C03601=1034.717,46.455,-90.669,168.917,41.159,157.714
C03602=1034.724,46.704,-90.686,168.919,41.158,157.713
C03603=1034.729,46.954,-90.702,168.921,41.158,157.714
C03604=1034.735,47.203,-90.720,168.923,41.158,157.714
C03605=1034.742,47.452,-90.737,168.926,41.157,157.714
C03606=1034.748,47.701,-90.753,168.928,41.156,157.714
C03607=1034.754,47.951,-90.771,168.930,41.156,157.714
C03608=1034.760,48.200,-90.788,168.932,41.156,157.714
C03609=1034.767,48.450,-90.805,168.934,41.156,157.714
C03610=1034.773,48.699,-90.822,168.937,41.155,157.714
C03611=1034.779,48.948,-90.840,168.939,41.154,157.714
C03612=1034.785,49.198,-90.856,168.941,41.154,157.714
C03613=1034.791,49.447,-90.873,168.943,41.154,157.714
C03614=1034.797,49.696,-90.891,168.945,41.153,157.714
C03615=1034.804,49.945,-90.908,168.947,41.153,157.714
C03616=1034.810,50.195,-90.925,168.950,41.152,157.714
C03617=1034.816,50.444,-90.942,168.951,41.151,157.714
C03618=1034.823,50.694,-90.960,168.953,41.151,157.714
C03619=1034.829,50.942,-90.977,168.956,41.151,157.714
C03620=1034.835,51.192,-90.993,168.958,41.151,157.714
C03621=1034.841,51.441,-91.011,168.960,41.150,157.714
C03622=1034.848,51.691,-91.028,168.962,41.149,157.714
C03623=1034.854,51.940,-91.045,168.964,41.149,157.714
C03624=1034.860,52.190,-91.062,168.966,41.148,157.714
C03625=1034.867,52.439,-91.080,168.968,41.148,157.714
C03626=1034.873,52.688,-91.097,168.971,41.148,157.714
C03627=1034.879,52.938,-91.115,168.973,41.147,157.714
C03628=1034.885,53.187,-91.131,168.975,41.147,157.714
C03629=1034.892,53.437,-91.148,168.977,41.146,157.714
C03630=1034.897,53.686,-91.166,168.979,41.146,157.714
C03631=1034.904,53.935,-91.183,168.982,41.145,157.714
C03632=1034.911,54.184,-91.200,168.984,41.145,157.714
C03633=1034.917,54.433,-91.218,168.986,41.145,157.715
C03634=1034.923,54.682,-91.235,168.988,41.144,157.714
C03635=1034.929,54.932,-91.252,168.990,41.143,157.715
C03636=1034.936,55.182,-91.269,168.993,41.143,157.715
C03637=1034.942,55.431,-91.286,168.995,41.142,157.715
C03638=1034.949,55.680,-91.304,168.997,41.142,157.715
C03639=1034.955,55.929,-91.321,168.999,41.142,157.715
C03640=1034.961,56.179,-91.339,169.001,41.141,157.715
C03641=1034.968,56.428,-91.356,169.004,41.140,157.715
C03642=1034.974,56.677,-91.373,169.006,41.140,157.715
C03643=1034.980,56.927,-91.390,169.008,41.139,157.715
C03644=1034.986,57.176,-91.407,169.010,41.139,157.715
C03645=1034.993,57.425,-91.424,169.012,41.139,157.715
C03646=1034.999,57.675,-91.442,169.015,41.138,157.715
C03647=1035.006,57.924,-91.459,169.017,41.138,157.715
C03648=1035.012,58.174,-91.477,169.019,41.137,157.715
C03649=1035.018,58.423,-91.495,169.021,41.136,157.715
C03650=1035.025,58.672,-91.512,169.023,41.136,157.715
C03651=1035.031,58.921,-91.530,169.026,41.136,157.715
C03652=1035.038,59.171,-91.547,169.028,41.135,157.715
C03653=1035.044,59.420,-91.564,169.030,41.135,157.715
C03654=1035.050,59.669,-91.582,169.032,41.134,157.715
C03655=1035.056,59.918,-91.599,169.034,41.134,157.715
C03656=1035.064,60.205,-91.619,169.037,41.133,157.715
C03657=1035.071,60.491,-91.639,169.039,41.132,157.715
C03658=1035.079,60.777,-91.659,169.041,41.132,157.715
C03659=1035.086,61.063,-91.679,169.044,41.131,157.715
C03660=1035.092,61.313,-91.697,169.046,41.131,157.715
C03661=1035.099,61.561,-91.714,169.048,41.130,157.715
C03662=1035.105,61.811,-91.731,169.050,41.130,157.715
C03663=1035.112,62.061,-91.749,169.052,41.129,157.715
C03664=1035.118,62.310,-91.766,169.055,41.128,157.715
C03665=1035.125,62.558,-91.784,169.057,41.128,157.715
C03666=1035.131,62.808,-91.802,169.059,41.128,157.715
C03667=1035.138,63.057,-91.819,169.061,41.127,157.715
C03668=1035.144,63.306,-91.836,169.064,41.127,157.715
C03669=1035.150,63.556,-91.854,169.066,41.126,157.715
C03670=1035.157,63.805,-91.871,169.068,41.125,157.715
C03671=1035.163,64.055,-91.889,169.070,41.125,157.715
C03672=1035.169,64.304,-91.907,169.072,41.125,157.715
C03673=1035.176,64.553,-91.925,169.074,41.124,157.715
C03674=1035.182,64.802,-91.943,169.077,41.124,157.715
C03675=1035.188,65.052,-91.961,169.079,41.123,157.715
C03676=1035.194,65.301,-91.978,169.081,41.123,157.716
C03677=1035.201,65.551,-91.996,169.083,41.122,157.715
C03678=1035.208,65.800,-92.014,169.085,41.122,157.716
C03679=1035.213,66.049,-92.031,169.088,41.122,157.716
C03680=1035.219,66.298,-92.049,169.090,41.122,157.716
C03681=1035.226,66.548,-92.067,169.092,41.121,157.716
C03682=1035.232,66.796,-92.085,169.094,41.120,157.716
C03683=1035.238,67.046,-92.103,169.096,41.120,157.716
C03684=1035.245,67.295,-92.120,169.098,41.120,157.716
C03685=1035.251,67.544,-92.139,169.101,41.119,157.716
C03686=1035.257,67.793,-92.156,169.103,41.119,157.716
C03687=1035.263,68.043,-92.174,169.105,41.118,157.716
C03688=1035.270,68.292,-92.192,169.107,41.118,157.716
C03689=1035.276,68.542,-92.210,169.109,41.117,157.716
C03690=1035.282,68.791,-92.228,169.111,41.117,157.716
C03691=1035.289,69.040,-92.246,169.114,41.117,157.716
C03692=1035.295,69.289,-92.264,169.116,41.116,157.716
C03693=1035.301,69.539,-92.282,169.118,41.116,157.716
C03694=1035.308,69.788,-92.300,169.120,41.115,157.716
C03695=1035.313,70.037,-92.318,169.122,41.115,157.716
C03696=1035.320,70.287,-92.335,169.124,41.115,157.716
C03697=1035.327,70.536,-92.354,169.127,41.114,157.716
C03698=1035.333,70.786,-92.372,169.129,41.114,157.716
C03699=1035.338,71.034,-92.390,169.131,41.113,157.716
C03700=1035.345,71.284,-92.408,169.133,41.113,157.716
C03701=1035.351,71.533,-92.427,169.135,41.113,157.716
C03702=1035.357,71.783,-92.445,169.137,41.113,157.716
C03703=1035.364,72.031,-92.463,169.140,41.112,157.717
C03704=1035.370,72.280,-92.480,169.142,41.111,157.716
C03705=1035.376,72.530,-92.498,169.144,41.111,157.717
C03706=1035.382,72.779,-92.517,169.146,41.111,157.717
C03707=1035.388,73.029,-92.535,169.148,41.111,157.717
C03708=1035.395,73.278,-92.554,169.150,41.110,157.717
C03709=1035.400,73.527,-92.571,169.152,41.110,157.717
C03710=1035.408,73.776,-92.589,169.155,41.109,157.717
C03711=1035.414,74.025,-92.608,169.157,41.109,157.717
C03712=1035.420,74.275,-92.626,169.159,41.109,157.717
C03713=1035.427,74.524,-92.644,169.161,41.108,157.717
C03714=1035.433,74.774,-92.662,169.163,41.108,157.717
C03715=1035.439,75.022,-92.681,169.165,41.107,157.717
C03716=1035.445,75.272,-92.699,169.168,41.107,157.717
C03717=1035.451,75.521,-92.717,169.170,41.107,157.717
C03718=1035.457,75.771,-92.735,169.172,41.106,157.717
C03719=1035.464,76.020,-92.753,169.174,41.106,157.717
C03720=1035.471,76.305,-92.774,169.177,41.105,157.717
C03721=1035.479,76.591,-92.795,169.179,41.105,157.717
C03722=1035.485,76.877,-92.816,169.182,41.104,157.717
C03723=1035.493,77.163,-92.837,169.184,41.104,157.717
C03724=1035.499,77.413,-92.856,169.186,41.103,157.717
C03725=1035.506,77.662,-92.874,169.188,41.103,157.717
C03726=1035.511,77.911,-92.892,169.191,41.103,157.717
C03727=1035.518,78.160,-92.911,169.193,41.103,157.717
C03728=1035.524,78.409,-92.929,169.195,41.102,157.717
C03729=1035.530,78.659,-92.947,169.197,41.102,157.717
C03730=1035.536,78.908,-92.966,169.199,41.101,157.718
C03731=1035.542,79.157,-92.985,169.201,41.101,157.718
C03732=1035.548,79.407,-93.003,169.203,41.101,157.718
C03733=1035.555,79.656,-93.022,169.206,41.100,157.718
C03734=1035.561,79.905,-93.040,169.208,41.100,157.718
C03735=1035.567,80.154,-93.059,169.210,41.100,157.718
C03736=1035.573,80.403,-93.077,169.212,41.100,157.718
C03737=1035.579,80.653,-93.096,169.214,41.099,157.718
C03738=1035.585,80.902,-93.114,169.216,41.099,157.718
C03739=1035.592,81.151,-93.133,169.218,41.098,157.718
C03740=1035.598,81.400,-93.152,169.221,41.098,157.718
C03741=1035.604,81.650,-93.170,169.223,41.098,157.718
C03742=1035.611,81.899,-93.188,169.225,41.097,157.718
C03743=1035.616,82.149,-93.208,169.227,41.097,157.718
C03744=1035.623,82.398,-93.226,169.229,41.097,157.718
C03745=1035.629,82.646,-93.244,169.231,41.096,157.718
C03746=1035.635,82.895,-93.263,169.233,41.096,157.718
C03747=1035.641,83.145,-93.281,169.236,41.096,157.718
C03748=1035.648,83.394,-93.300,169.238,41.095,157.718
C03749=1035.653,83.643,-93.319,169.240,41.095,157.719
C03750=1035.660,83.893,-93.338,169.242,41.095,157.719
C03751=1035.666,84.142,-93.356,169.244,41.095,157.719
C03752=1035.673,84.391,-93.375,169.246,41.094,157.719
C03753=1035.679,84.640,-93.394,169.249,41.093,157.719
C03754=1035.685,84.889,-93.412,169.251,41.093,157.719
C03755=1035.691,85.139,-93.431,169.253,41.093,157.719
C03756=1035.697,85.388,-93.449,169.255,41.093,157.719
C03757=1035.704,85.637,-93.468,169.257,41.092,157.719
C03758=1035.710,85.887,-93.487,169.259,41.091,157.719
C03759=1035.717,86.136,-93.505,169.262,41.091,157.719
C03760=1035.722,86.385,-93.525,169.264,41.091,157.719
C03761=1035.729,86.634,-93.543,169.266,41.091,157.719
C03762=1035.735,86.883,-93.562,169.268,41.090,157.719
C03763=1035.742,87.132,-93.580,169.270,41.090,157.719
C03764=1035.748,87.382,-93.599,169.272,41.089,157.719
C03765=1035.754,87.631,-93.618,169.275,41.089,157.719
C03766=1035.760,87.880,-93.637,169.277,41.089,157.719
C03767=1035.766,88.129,-93.656,169.279,41.088,157.719
C03768=1035.773,88.378,-93.674,169.281,41.088,157.719
C03769=1035.779,88.627,-93.693,169.283,41.087,157.719
C03770=1035.786,88.877,-93.712,169.286,41.087,157.719
C03771=1035.791,89.126,-93.731,169.288,41.087,157.719
C03772=1035.798,89.375,-93.750,169.290,41.086,157.719
C03773=1035.805,89.625,-93.769,169.292,41.086,157.720
C03774=1035.811,89.874,-93.787,169.294,41.085,157.719
C03775=1035.817,90.124,-93.806,169.296,41.085,157.720
C03776=1035.823,90.373,-93.825,169.299,41.085,157.720
C03777=1035.829,90.622,-93.844,169.301,41.084,157.720
C03778=1035.836,90.871,-93.864,169.303,41.084,157.720
C03779=1035.842,91.120,-93.883,169.305,41.084,157.720
C03780=1035.848,91.369,-93.902,169.307,41.084,157.720
C03781=1035.854,91.619,-93.921,169.309,41.084,157.720
C03782=1035.860,91.868,-93.939,169.311,41.083,157.720
C03783=1035.867,92.117,-93.958,169.314,41.083,157.720
C03784=1035.874,92.403,-93.980,169.316,41.083,157.720
C03785=1035.880,92.688,-94.002,169.319,41.082,157.720
C03786=1035.887,92.974,-94.025,169.321,41.082,157.720
C03787=1035.894,93.260,-94.046,169.324,41.082,157.720
C03788=1035.901,93.509,-94.066,169.326,41.081,157.720
C03789=1035.907,93.758,-94.085,169.328,41.081,157.721
C03790=1035.913,94.008,-94.104,169.330,41.080,157.720
C03791=1035.919,94.257,-94.123,169.332,41.080,157.720
C03792=1035.926,94.505,-94.142,169.334,41.080,157.721
C03793=1035.931,94.755,-94.161,169.336,41.080,157.721
C03794=1035.938,95.004,-94.180,169.339,41.079,157.721
C03795=1035.944,95.254,-94.200,169.341,41.079,157.721
C03796=1035.951,95.503,-94.219,169.343,41.079,157.721
C03797=1035.956,95.752,-94.238,169.345,41.079,157.721
C03798=1035.963,96.001,-94.257,169.347,41.078,157.721
C03799=1035.969,96.251,-94.276,169.349,41.078,157.721
C03800=1035.975,96.499,-94.296,169.352,41.078,157.721
C03801=1035.981,96.749,-94.315,169.354,41.077,157.721
C03802=1035.987,96.998,-94.333,169.356,41.077,157.721
C03803=1035.994,97.247,-94.354,169.358,41.076,157.721
C03804=1036.000,97.496,-94.372,169.360,41.076,157.721
C03805=1036.006,97.746,-94.392,169.363,41.076,157.721
C03806=1036.013,97.994,-94.411,169.365,41.076,157.721
C03807=1036.018,98.244,-94.430,169.367,41.075,157.721
C03808=1036.025,98.493,-94.449,169.369,41.075,157.721
C03809=1036.032,98.742,-94.469,169.371,41.075,157.722
C03810=1036.038,98.991,-94.488,169.373,41.075,157.722
C03811=1036.044,99.240,-94.508,169.376,41.074,157.722
C03812=1036.050,99.489,-94.526,169.378,41.073,157.722
C03813=1036.056,99.739,-94.546,169.380,41.073,157.722
C03814=1036.063,99.988,-94.565,169.382,41.073,157.722
C03815=1036.069,100.237,-94.585,169.384,41.073,157.722
C03816=1036.075,100.486,-94.605,169.387,41.072,157.722
C03817=1036.081,100.735,-94.623,169.389,41.072,157.722
C03818=1036.087,100.984,-94.643,169.391,41.072,157.722
C03819=1036.093,101.234,-94.662,169.393,41.071,157.722
C03820=1036.100,101.483,-94.683,169.395,41.071,157.722
C03821=1036.106,101.732,-94.701,169.397,41.071,157.722
C03822=1036.112,101.981,-94.721,169.400,41.071,157.722
C03823=1036.118,102.231,-94.741,169.402,41.070,157.722
C03824=1036.124,102.479,-94.761,169.404,41.070,157.722
C03825=1036.130,102.729,-94.780,169.406,41.070,157.722
C03826=1036.137,102.978,-94.800,169.408,41.070,157.722
C03827=1036.143,103.227,-94.820,169.411,41.069,157.723
C03828=1036.149,103.476,-94.839,169.414,41.069,157.723
C03829=1036.155,103.725,-94.859,169.416,41.069,157.723
C03830=1036.161,103.974,-94.877,169.418,41.069,157.723
C03831=1036.168,104.224,-94.898,169.420,41.068,157.723
C03832=1036.174,104.472,-94.918,169.422,41.068,157.723
C03833=1036.179,104.722,-94.937,169.424,41.068,157.723
C03834=1036.185,104.971,-94.957,169.427,41.068,157.723
C03835=1036.192,105.221,-94.976,169.429,41.067,157.723
C03836=1036.198,105.469,-94.996,169.431,41.067,157.723
C03837=1036.204,105.718,-95.016,169.433,41.067,157.723
C03838=1036.210,105.968,-95.035,169.435,41.067,157.723
C03839=1036.217,106.217,-95.055,169.438,41.066,157.723
C03840=1036.223,106.466,-95.075,169.440,41.066,157.723
C03841=1036.229,106.715,-95.094,169.442,41.066,157.723
C03842=1036.235,106.964,-95.114,169.444,41.066,157.724
C03843=1036.242,107.213,-95.134,169.446,41.065,157.724
C03844=1036.247,107.463,-95.154,169.448,41.065,157.724
C03845=1036.254,107.711,-95.173,169.451,41.065,157.724
C03846=1036.261,107.961,-95.193,169.453,41.064,157.724
C03847=1036.267,108.210,-95.213,169.455,41.064,157.724
C03848=1036.274,108.495,-95.236,169.458,41.064,157.724
C03849=1036.281,108.781,-95.258,169.460,41.064,157.724
C03850=1036.288,109.067,-95.281,169.463,41.063,157.724
C03851=1036.295,109.353,-95.304,169.465,41.063,157.724
C03852=1036.301,109.602,-95.324,169.467,41.063,157.724
C03853=1036.308,109.852,-95.343,169.470,41.062,157.724
C03854=1036.314,110.101,-95.363,169.472,41.062,157.724
C03855=1036.320,110.349,-95.383,169.474,41.062,157.724
C03856=1036.326,110.599,-95.403,169.476,41.062,157.724
C03857=1036.332,110.848,-95.423,169.478,41.061,157.725
C03858=1036.338,111.097,-95.442,169.481,41.061,157.725
C03859=1036.345,111.347,-95.462,169.483,41.061,157.725
C03860=1036.351,111.595,-95.482,169.485,41.061,157.725
C03861=1036.357,111.844,-95.502,169.487,41.060,157.725
C03862=1036.363,112.094,-95.523,169.489,41.060,157.725
C03863=1036.369,112.343,-95.543,169.492,41.060,157.725
C03864=1036.375,112.591,-95.563,169.495,41.060,157.725
C03865=1036.382,112.841,-95.583,169.497,41.059,157.725
C03866=1036.388,113.090,-95.602,169.499,41.059,157.725
C03867=1036.394,113.340,-95.623,169.501,41.059,157.725
C03868=1036.400,113.589,-95.642,169.504,41.058,157.725
C03869=1036.406,113.837,-95.662,169.506,41.058,157.725
C03870=1036.412,114.087,-95.683,169.508,41.058,157.725
C03871=1036.418,114.336,-95.703,169.510,41.058,157.726
C03872=1036.424,114.585,-95.723,169.512,41.058,157.726
C03873=1036.430,114.834,-95.743,169.515,41.058,157.726
C03874=1036.436,115.084,-95.764,169.517,41.058,157.726
C03875=1036.442,115.332,-95.784,169.519,41.057,157.726
C03876=1036.449,115.581,-95.805,169.521,41.057,157.726
C03877=1036.455,115.830,-95.825,169.523,41.057,157.726
C03878=1036.460,116.079,-95.846,169.525,41.057,157.726
C03879=1036.467,116.329,-95.866,169.528,41.057,157.726
C03880=1036.473,116.578,-95.886,169.530,41.057,157.726
C03881=1036.479,116.826,-95.906,169.532,41.056,157.726
C03882=1036.484,117.076,-95.927,169.534,41.056,157.726
C03883=1036.490,117.325,-95.947,169.536,41.057,157.727
C03884=1036.496,117.574,-95.967,169.540,41.056,157.727
C03885=1036.503,117.823,-95.987,169.542,41.056,157.727
C03886=1036.508,118.072,-96.008,169.544,41.056,157.727
C03887=1036.515,118.321,-96.029,169.546,41.055,157.727
C03888=1036.521,118.570,-96.049,169.548,41.055,157.727
C03889=1036.527,118.819,-96.069,169.551,41.055,157.727
C03890=1036.533,119.069,-96.090,169.553,41.055,157.727
C03891=1036.539,119.318,-96.109,169.555,41.055,157.727
C03892=1036.546,119.567,-96.130,169.557,41.055,157.727
C03893=1036.552,119.815,-96.150,169.559,41.055,157.727
C03894=1036.558,120.065,-96.171,169.562,41.054,157.727
C03895=1036.564,120.314,-96.191,169.564,41.054,157.728
C03896=1036.570,120.563,-96.212,169.566,41.054,157.728
C03897=1036.576,120.813,-96.232,169.568,41.053,157.728
C03898=1036.582,121.061,-96.253,169.571,41.054,157.728
C03899=1036.589,121.310,-96.273,169.573,41.054,157.728
C03900=1036.595,121.559,-96.293,169.575,41.053,157.728
C03901=1036.600,121.809,-96.314,169.577,41.053,157.728
C03902=1036.606,122.058,-96.334,169.579,41.053,157.728
C03903=1036.613,122.307,-96.355,169.582,41.052,157.728
C03904=1036.619,122.556,-96.376,169.584,41.052,157.728
C03905=1036.625,122.805,-96.396,169.586,41.052,157.728
C03906=1036.631,123.053,-96.417,169.589,41.052,157.729
C03907=1036.638,123.303,-96.437,169.592,41.052,157.729
C03908=1036.643,123.552,-96.458,169.594,41.052,157.729
C03909=1036.650,123.802,-96.478,169.596,41.052,157.729
C03910=1036.656,124.050,-96.499,169.598,41.051,157.729
C03911=1036.662,124.300,-96.519,169.601,41.051,157.729
C03912=1036.669,124.585,-96.543,169.603,41.051,157.729
C03913=1036.676,124.870,-96.567,169.606,41.050,157.729
C03914=1036.683,125.156,-96.590,169.608,41.051,157.729
C03915=1036.690,125.443,-96.614,169.611,41.050,157.729
C03916=1036.697,125.691,-96.634,169.613,41.050,157.729
C03917=1036.703,125.940,-96.655,169.615,41.050,157.729
C03918=1036.709,126.189,-96.675,169.618,41.050,157.729
C03919=1036.715,126.438,-96.696,169.620,41.049,157.730
C03920=1036.722,126.688,-96.717,169.622,41.049,157.730
C03921=1036.728,126.936,-96.737,169.625,41.049,157.730
C03922=1036.734,127.186,-96.758,169.627,41.048,157.730
C03923=1036.740,127.435,-96.778,169.629,41.048,157.730
C03924=1036.747,127.684,-96.799,169.631,41.049,157.730
C03925=1036.752,127.933,-96.820,169.634,41.048,157.730
C03926=1036.759,128.182,-96.841,169.636,41.048,157.730
C03927=1036.766,128.431,-96.861,169.638,41.048,157.730
C03928=1036.771,128.680,-96.882,169.642,41.047,157.730
C03929=1036.778,128.929,-96.903,169.644,41.047,157.730
C03930=1036.785,129.179,-96.923,169.646,41.047,157.730
C03931=1036.790,129.427,-96.944,169.648,41.047,157.730
C03932=1036.797,129.677,-96.965,169.651,41.046,157.731
C03933=1036.803,129.925,-96.985,169.653,41.046,157.731
C03934=1036.809,130.175,-97.006,169.655,41.046,157.731
C03935=1036.816,130.424,-97.027,169.658,41.046,157.731
C03936=1036.822,130.672,-97.047,169.660,41.046,157.731
C03937=1036.828,130.922,-97.069,169.662,41.046,157.731
C03938=1036.835,131.170,-97.090,169.664,41.045,157.731
C03939=1036.840,131.420,-97.111,169.667,41.045,157.731
C03940=1036.846,131.669,-97.132,169.669,41.045,157.731
C03941=1036.852,131.918,-97.152,169.671,41.045,157.731
C03942=1036.858,132.167,-97.174,169.673,41.045,157.731
C03943=1036.865,132.416,-97.195,169.676,41.045,157.732
C03944=1036.871,132.665,-97.215,169.678,41.044,157.732
C03945=1036.877,132.914,-97.237,169.680,41.045,157.732
C03946=1036.884,133.163,-97.258,169.683,41.044,157.732
C03947=1036.889,133.412,-97.279,169.685,41.044,157.732
C03948=1036.895,133.661,-97.300,169.688,41.044,157.732
C03949=1036.901,133.909,-97.321,169.690,41.044,157.732
C03950=1036.907,134.159,-97.342,169.693,41.044,157.732
C03951=1036.913,134.408,-97.363,169.695,41.044,157.732
C03952=1036.920,134.657,-97.384,169.697,41.043,157.732
C03953=1036.926,134.906,-97.406,169.700,41.044,157.733
C03954=1036.932,135.156,-97.427,169.702,41.044,157.733
C03955=1036.938,135.404,-97.447,169.704,41.043,157.733
C03956=1036.944,135.653,-97.469,169.706,41.043,157.733
C03957=1036.951,135.902,-97.490,169.709,41.043,157.733
C03958=1036.957,136.152,-97.511,169.711,41.043,157.733
C03959=1036.962,136.400,-97.532,169.713,41.043,157.733
C03960=1036.969,136.649,-97.553,169.716,41.042,157.733
C03961=1036.976,136.898,-97.575,169.719,41.043,157.733
C03962=1036.981,137.147,-97.596,169.721,41.043,157.733
C03963=1036.987,137.397,-97.617,169.724,41.042,157.734
C03964=1036.994,137.646,-97.638,169.726,41.042,157.734
C03965=1036.999,137.894,-97.659,169.728,41.042,157.734
C03966=1037.006,138.143,-97.681,169.730,41.042,157.734
C03967=1037.012,138.393,-97.703,169.733,41.042,157.734
C03968=1037.019,138.641,-97.724,169.735,41.042,157.734
C03969=1037.024,138.891,-97.744,169.737,41.042,157.734
C03970=1037.030,139.140,-97.766,169.740,41.042,157.734
C03971=1037.036,139.389,-97.788,169.742,41.041,157.734
C03972=1037.042,139.638,-97.809,169.744,41.042,157.735
C03973=1037.049,139.886,-97.830,169.747,41.041,157.735
C03974=1037.055,140.136,-97.851,169.749,41.041,157.735
C03975=1037.061,140.385,-97.873,169.752,41.042,157.735
C03976=1037.068,140.670,-97.898,169.755,41.041,157.735
C03977=1037.075,140.955,-97.922,169.758,41.042,157.735
C03978=1037.082,141.241,-97.947,169.760,41.041,157.735
C03979=1037.088,141.526,-97.972,169.763,41.041,157.735
C03980=1037.095,141.775,-97.994,169.765,41.041,157.736
C03981=1037.101,142.025,-98.015,169.767,41.041,157.736
C03982=1037.108,142.273,-98.036,169.770,41.041,157.736
C03983=1037.113,142.522,-98.058,169.772,41.041,157.736
C03984=1037.119,142.771,-98.079,169.774,41.041,157.736
C03985=1037.125,143.020,-98.101,169.777,41.041,157.736
C03986=1037.132,143.270,-98.122,169.780,41.041,157.736
C03987=1037.137,143.518,-98.144,169.782,41.041,157.736
C03988=1037.143,143.767,-98.165,169.785,41.041,157.736
C03989=1037.150,144.016,-98.187,169.787,41.041,157.737
C03990=1037.156,144.266,-98.209,169.789,41.040,157.737
C03991=1037.162,144.515,-98.230,169.792,41.041,157.737
C03992=1037.168,144.764,-98.252,169.794,41.041,157.737
C03993=1037.174,145.012,-98.274,169.797,41.040,157.737
C03994=1037.181,145.261,-98.295,169.799,41.041,157.737
C03995=1037.187,145.510,-98.317,169.801,41.040,157.737
C03996=1037.193,145.759,-98.338,169.804,41.040,157.737
C03997=1037.199,146.008,-98.360,169.806,41.040,157.737
C03998=1037.205,146.258,-98.382,169.808,41.040,157.738
C03999=1037.211,146.506,-98.403,169.812,41.040,157.738
C04000=1037.217,146.755,-98.425,169.814,41.040,157.738
C04001=1037.224,147.004,-98.447,169.816,41.040,157.738
C04002=1037.230,147.253,-98.468,169.819,41.040,157.738
C04003=1037.236,147.502,-98.490,169.821,41.040,157.738
C04004=1037.242,147.751,-98.512,169.823,41.040,157.738
C04005=1037.249,148.000,-98.534,169.826,41.040,157.738
C04006=1037.253,148.249,-98.556,169.828,41.040,157.738
C04007=1037.260,148.498,-98.578,169.831,41.040,157.739
C04008=1037.266,148.747,-98.600,169.833,41.040,157.739
C04009=1037.272,148.996,-98.622,169.836,41.040,157.739
C04010=1037.278,149.245,-98.643,169.839,41.040,157.739
C04011=1037.285,149.494,-98.665,169.841,41.040,157.739
C04012=1037.291,149.743,-98.687,169.843,41.040,157.739
C04013=1037.296,149.993,-98.709,169.846,41.040,157.739
C04014=1037.302,150.240,-98.731,169.848,41.040,157.740
C04015=1037.308,150.490,-98.753,169.850,41.040,157.740
C04016=1037.315,150.739,-98.775,169.853,41.040,157.740
C04017=1037.321,150.987,-98.797,169.855,41.040,157.740
C04018=1037.327,151.237,-98.819,169.859,41.040,157.740
C04019=1037.333,151.485,-98.842,169.861,41.040,157.740
C04020=1037.339,151.735,-98.863,169.863,41.040,157.740
C04021=1037.345,151.984,-98.885,169.866,41.040,157.740
C04022=1037.352,152.232,-98.907,169.868,41.040,157.741
C04023=1037.358,152.482,-98.929,169.870,41.040,157.741
C04024=1037.364,152.731,-98.952,169.873,41.040,157.741
C04025=1037.370,152.980,-98.973,169.875,41.040,157.741
C04026=1037.376,153.228,-98.995,169.878,41.040,157.741
C04027=1037.382,153.477,-99.017,169.880,41.040,157.741
C04028=1037.388,153.726,-99.039,169.883,41.041,157.741
C04029=1037.394,153.975,-99.062,169.886,41.040,157.742
C04030=1037.400,154.224,-99.083,169.888,41.040,157.742
C04031=1037.406,154.473,-99.106,169.891,41.040,157.742
C04032=1037.414,154.794,-99.134,169.894,41.040,157.742
C04033=1037.422,155.115,-99.164,169.897,41.040,157.742
C04034=1037.430,155.437,-99.192,169.900,41.040,157.742
C04035=1037.438,155.758,-99.220,169.903,41.041,157.743
C04036=1037.443,155.989,-99.241,169.905,41.040,157.743
C04037=1037.449,156.219,-99.262,169.909,41.041,157.743
C04038=1037.454,156.450,-99.282,169.911,41.040,157.743
C04039=1037.460,156.682,-99.303,169.913,41.041,157.743
C04040=1037.466,156.912,-99.324,169.915,41.041,157.743
C04041=1037.471,157.143,-99.344,169.917,41.041,157.743
C04042=1037.478,157.374,-99.365,169.920,41.041,157.743
C04043=1037.483,157.605,-99.386,169.922,41.041,157.744
C04044=1037.489,157.854,-99.408,169.924,41.041,157.744
C04045=1037.495,158.103,-99.431,169.928,41.041,157.744
C04046=1037.501,158.351,-99.453,169.930,41.041,157.744
C04047=1037.507,158.601,-99.475,169.933,41.041,157.744
C04048=1037.513,158.850,-99.498,169.935,41.042,157.744
C04049=1037.520,159.098,-99.520,169.938,41.041,157.744
C04050=1037.525,159.348,-99.542,169.940,41.042,157.745
C04051=1037.532,159.596,-99.564,169.942,41.041,157.745
C04052=1037.538,159.845,-99.587,169.945,41.042,157.745
C04053=1037.545,160.094,-99.610,169.947,41.041,157.745
C04054=1037.550,160.344,-99.632,169.951,41.042,157.745
C04055=1037.556,160.593,-99.655,169.953,41.042,157.745
C04056=1037.562,160.841,-99.678,169.956,41.042,157.746
C04057=1037.568,161.090,-99.701,169.958,41.043,157.746
C04058=1037.574,161.339,-99.724,169.960,41.042,157.746
C04059=1037.580,161.588,-99.746,169.963,41.043,157.746
C04060=1037.586,161.837,-99.769,169.966,41.043,157.746
C04061=1037.592,162.086,-99.792,169.969,41.043,157.747
C04062=1037.597,162.334,-99.815,169.971,41.043,157.747
C04063=1037.603,162.584,-99.837,169.973,41.044,157.747
C04064=1037.609,162.833,-99.859,169.976,41.044,157.747
C04065=1037.615,163.081,-99.882,169.978,41.044,157.747
C04066=1037.621,163.330,-99.905,169.982,41.044,157.747
C04067=1037.626,163.579,-99.928,169.984,41.044,157.747
C04068=1037.633,163.828,-99.951,169.986,41.045,157.748
C04069=1037.639,164.077,-99.973,169.989,41.045,157.748
C04070=1037.644,164.326,-99.996,169.991,41.045,157.748
C04071=1037.650,164.575,-100.019,169.994,41.046,157.748
C04072=1037.656,164.823,-100.042,169.996,41.045,157.748
C04073=1037.662,165.072,-100.065,170.000,41.046,157.749
C04074=1037.668,165.321,-100.088,170.002,41.046,157.749
C04075=1037.674,165.571,-100.111,170.005,41.046,157.749
C04076=1037.680,165.819,-100.134,170.007,41.046,157.749
C04077=1037.686,166.068,-100.158,170.009,41.046,157.749
C04078=1037.693,166.316,-100.180,170.012,41.047,157.749
C04079=1037.698,166.565,-100.203,170.015,41.047,157.750
C04080=1037.704,166.814,-100.226,170.018,41.047,157.750
C04081=1037.710,167.063,-100.249,170.020,41.047,157.750
C04082=1037.715,167.312,-100.272,170.023,41.047,157.750
C04083=1037.723,167.561,-100.294,170.025,41.048,157.750
C04084=1037.728,167.810,-100.317,170.028,41.048,157.751
C04085=1037.734,168.059,-100.340,170.031,41.048,157.751
C04086=1037.740,168.308,-100.363,170.034,41.048,157.751
C04087=1037.746,168.556,-100.387,170.036,41.048,157.751
C04088=1037.752,168.805,-100.409,170.039,41.049,157.751
C04089=1037.759,169.054,-100.433,170.041,41.049,157.751
C04090=1037.764,169.303,-100.455,170.044,41.049,157.752
C04091=1037.770,169.552,-100.478,170.046,41.049,157.752
C04092=1037.776,169.800,-100.502,170.050,41.049,157.752
C04093=1037.782,170.049,-100.525,170.052,41.050,157.752
C04094=1037.789,170.299,-100.548,170.055,41.050,157.752
C04095=1037.795,170.547,-100.571,170.057,41.051,157.753
C04096=1037.800,170.796,-100.594,170.060,41.051,157.753
C04097=1037.806,171.045,-100.617,170.062,41.051,157.753
C04098=1037.812,171.294,-100.640,170.066,41.051,157.753
C04099=1037.818,171.543,-100.664,170.068,41.051,157.753
C04100=1037.825,171.792,-100.686,170.071,41.051,157.753
C04101=1037.831,172.040,-100.710,170.073,41.052,157.754
C04102=1037.837,172.290,-100.733,170.076,41.052,157.754
C04103=1037.843,172.538,-100.756,170.078,41.052,157.754
C04104=1037.850,172.822,-100.782,170.082,41.052,157.754
C04105=1037.857,173.108,-100.809,170.085,41.052,157.754
C04106=1037.864,173.392,-100.835,170.088,41.053,157.755
C04107=1037.871,173.677,-100.862,170.091,41.053,157.755
C04108=1037.877,173.925,-100.886,170.094,41.053,157.755
C04109=1037.883,174.175,-100.909,170.097,41.054,157.755
C04110=1037.890,174.424,-100.931,170.100,41.054,157.755
C04111=1037.896,174.672,-100.955,170.102,41.054,157.755
C04112=1037.901,174.921,-100.978,170.105,41.054,157.756
C04113=1037.908,175.170,-101.002,170.107,41.054,157.756
C04114=1037.914,175.419,-101.025,170.110,41.055,157.756
C04115=1037.920,175.667,-101.048,170.114,41.055,157.756
C04116=1037.926,175.916,-101.072,170.116,41.055,157.757
C04117=1037.933,176.165,-101.094,170.119,41.055,157.757
C04118=1037.939,176.414,-101.118,170.121,41.055,157.757
C04119=1037.945,176.663,-101.141,170.124,41.056,157.757
C04120=1037.951,176.911,-101.165,170.127,41.056,157.757
C04121=1037.957,177.161,-101.188,170.130,41.056,157.757
C04122=1037.963,177.409,-101.212,170.133,41.057,157.758
C04123=1037.969,177.658,-101.235,170.135,41.057,157.758
C04124=1037.977,177.907,-101.258,170.138,41.057,157.758
C04125=1037.982,178.156,-101.281,170.141,41.057,157.758
C04126=1037.989,178.405,-101.305,170.143,41.057,157.758
C04127=1037.995,178.653,-101.328,170.147,41.057,157.759
C04128=1038.001,178.902,-101.352,170.149,41.058,157.759
C04129=1038.007,179.151,-101.375,170.152,41.058,157.759
C04130=1038.013,179.400,-101.399,170.155,41.058,157.759
C04131=1038.019,179.649,-101.422,170.157,41.059,157.759
C04132=1038.025,179.897,-101.446,170.160,41.058,157.759
C04133=1038.033,180.146,-101.469,170.164,41.059,157.760
C04134=1038.039,180.395,-101.492,170.166,41.059,157.760
C04135=1038.045,180.644,-101.516,170.169,41.059,157.760
C04136=1038.051,180.893,-101.539,170.171,41.060,157.760
C04137=1038.058,181.142,-101.563,170.174,41.060,157.761
C04138=1038.064,181.390,-101.587,170.177,41.060,157.761
C04139=1038.070,181.640,-101.610,170.180,41.061,157.761
C04140=1038.076,181.888,-101.634,170.183,41.060,157.761
C04141=1038.083,182.137,-101.658,170.186,41.061,157.761
C04142=1038.088,182.386,-101.681,170.188,41.061,157.761
C04143=1038.096,182.635,-101.704,170.191,41.061,157.762
C04144=1038.102,182.883,-101.728,170.194,41.061,157.762
C04145=1038.108,183.132,-101.751,170.197,41.062,157.762
C04146=1038.114,183.381,-101.775,170.200,41.062,157.762
C04147=1038.120,183.630,-101.799,170.203,41.062,157.763
C04148=1038.126,183.878,-101.823,170.205,41.063,157.763
C04149=1038.133,184.127,-101.847,170.208,41.063,157.763
C04150=1038.138,184.376,-101.871,170.212,41.064,157.763
C04151=1038.144,184.624,-101.895,170.214,41.064,157.763
C04152=1038.150,184.873,-101.920,170.217,41.065,157.764
C04153=1038.156,185.122,-101.943,170.219,41.065,157.764
C04154=1038.162,185.372,-101.967,170.223,41.066,157.764
C04155=1038.168,185.620,-101.991,170.226,41.066,157.764
C04156=1038.173,185.869,-102.015,170.228,41.067,157.765
C04157=1038.180,186.117,-102.039,170.231,41.067,157.765
C04158=1038.185,186.367,-102.064,170.234,41.067,157.765
C04159=1038.191,186.615,-102.087,170.237,41.068,157.765
C04160=1038.197,186.864,-102.112,170.240,41.068,157.766
C04161=1038.203,187.113,-102.136,170.242,41.069,157.766
C04162=1038.209,187.362,-102.160,170.245,41.069,157.766
C04163=1038.215,187.610,-102.184,170.249,41.070,157.766
C04164=1038.222,187.859,-102.209,170.251,41.070,157.767
C04165=1038.228,188.107,-102.233,170.254,41.071,157.767
C04166=1038.233,188.356,-102.258,170.257,41.071,157.767
C04167=1038.240,188.605,-102.281,170.260,41.072,157.767
C04168=1038.247,188.889,-102.309,170.263,41.072,157.768
C04169=1038.253,189.173,-102.336,170.266,41.073,157.768
C04170=1038.260,189.458,-102.364,170.270,41.073,157.768
C04171=1038.267,189.742,-102.392,170.273,41.074,157.768
C04172=1038.273,189.991,-102.416,170.276,41.074,157.769
C04173=1038.279,190.240,-102.441,170.279,41.075,157.769
C04174=1038.285,190.488,-102.464,170.283,41.075,157.769
C04175=1038.291,190.737,-102.490,170.285,41.076,157.770
C04176=1038.298,190.986,-102.514,170.288,41.076,157.770
C04177=1038.303,191.234,-102.538,170.291,41.077,157.770
C04178=1038.310,191.483,-102.562,170.293,41.077,157.770
C04179=1038.315,191.732,-102.586,170.297,41.078,157.771
C04180=1038.322,191.980,-102.611,170.300,41.078,157.771
C04181=1038.328,192.230,-102.636,170.302,41.078,157.771
C04182=1038.334,192.478,-102.659,170.306,41.079,157.771
C04183=1038.340,192.727,-102.684,170.309,41.080,157.772
C04184=1038.347,192.976,-102.709,170.312,41.080,157.772
C04185=1038.352,193.224,-102.733,170.314,41.081,157.772
C04186=1038.359,193.473,-102.757,170.318,41.081,157.772
C04187=1038.365,193.722,-102.782,170.321,41.081,157.773
C04188=1038.371,193.970,-102.806,170.323,41.082,157.773
C04189=1038.377,194.219,-102.830,170.326,41.083,157.773
C04190=1038.384,194.468,-102.855,170.329,41.083,157.773
C04191=1038.389,194.716,-102.879,170.333,41.083,157.774
C04192=1038.396,194.965,-102.903,170.335,41.084,157.774
C04193=1038.402,195.214,-102.929,170.338,41.085,157.774
C04194=1038.409,195.463,-102.953,170.341,41.085,157.774
C04195=1038.414,195.712,-102.977,170.345,41.086,157.775
C04196=1038.420,195.960,-103.002,170.347,41.086,157.775
C04197=1038.427,196.209,-103.026,170.350,41.087,157.775
C04198=1038.432,196.457,-103.051,170.354,41.087,157.775
C04199=1038.439,196.706,-103.075,170.357,41.087,157.776
C04200=1038.445,196.955,-103.100,170.360,41.088,157.776
C04201=1038.452,197.204,-103.125,170.362,41.089,157.776
C04202=1038.458,197.453,-103.149,170.365,41.089,157.776
C04203=1038.464,197.701,-103.174,170.369,41.090,157.777
C04204=1038.470,197.950,-103.198,170.372,41.090,157.777
C04205=1038.476,198.199,-103.224,170.375,41.090,157.777
C04206=1038.483,198.448,-103.248,170.378,41.091,157.778
C04207=1038.488,198.696,-103.273,170.381,41.092,157.778
C04208=1038.495,198.945,-103.297,170.384,41.093,157.778
C04209=1038.501,199.193,-103.322,170.387,41.093,157.778
C04210=1038.508,199.442,-103.346,170.391,41.093,157.779
C04211=1038.514,199.691,-103.372,170.393,41.094,157.779
C04212=1038.521,199.940,-103.396,170.396,41.094,157.779
C04213=1038.526,200.188,-103.421,170.399,41.095,157.779
C04214=1038.533,200.437,-103.446,170.403,41.096,157.780
C04215=1038.539,200.686,-103.470,170.406,41.096,157.780
C04216=1038.545,200.934,-103.495,170.409,41.097,157.780
C04217=1038.552,201.183,-103.521,170.412,41.098,157.781
C04218=1038.557,201.432,-103.545,170.415,41.098,157.781
C04219=1038.564,201.681,-103.571,170.418,41.099,157.781
C04220=1038.570,201.928,-103.595,170.421,41.099,157.781
C04221=1038.576,202.178,-103.620,170.425,41.100,157.782
C04222=1038.582,202.426,-103.645,170.427,41.101,157.782
C04223=1038.588,202.675,-103.670,170.430,41.101,157.782
C04224=1038.595,202.924,-103.696,170.434,41.102,157.783
C04225=1038.601,203.172,-103.721,170.437,41.102,157.783
C04226=1038.606,203.421,-103.745,170.440,41.103,157.783
C04227=1038.612,203.670,-103.770,170.443,41.104,157.784
C04228=1038.618,203.918,-103.796,170.446,41.105,157.784
C04229=1038.625,204.167,-103.821,170.449,41.105,157.784
C04230=1038.631,204.416,-103.846,170.452,41.106,157.785
C04231=1038.638,204.664,-103.871,170.456,41.107,157.785
C04232=1038.663,205.715,-103.977,170.753,41.211,157.822
C04233=1038.672,206.029,-104.011,170.757,41.212,157.823
C04234=1038.681,206.344,-104.045,170.759,41.214,157.823
C04235=1038.690,206.658,-104.077,170.762,41.216,157.824
C04236=1038.698,206.973,-104.111,170.764,41.218,157.824
C04237=1038.704,207.221,-104.137,170.767,41.220,157.825
C04238=1038.711,207.470,-104.164,170.769,41.220,157.825
C04239=1038.718,207.718,-104.191,170.772,41.222,157.826
C04240=1038.725,207.966,-104.217,170.774,41.224,157.826
C04241=1038.731,208.215,-104.244,170.776,41.225,157.826
C04242=1038.738,208.463,-104.270,170.778,41.226,157.827
C04243=1038.745,208.712,-104.296,170.781,41.228,157.827
C04244=1038.751,208.961,-104.323,170.783,41.229,157.828
C04245=1038.758,209.209,-104.349,170.786,41.231,157.828
C04246=1038.765,209.458,-104.376,170.788,41.232,157.829
C04247=1038.771,209.707,-104.403,170.790,41.233,157.829
C04248=1038.778,209.954,-104.430,170.792,41.235,157.829
C04249=1038.785,210.203,-104.456,170.795,41.237,157.830
C04250=1038.791,210.451,-104.483,170.797,41.238,157.830
C04251=1038.798,210.700,-104.509,170.800,41.239,157.831
C04252=1038.805,210.949,-104.536,170.802,41.241,157.831
C04253=1038.811,211.197,-104.563,170.803,41.242,157.831
C04254=1038.818,211.445,-104.589,170.806,41.244,157.832
C04255=1038.825,211.695,-104.616,170.809,41.245,157.832
C04256=1038.831,211.943,-104.642,170.811,41.247,157.833
C04257=1038.838,212.191,-104.670,170.813,41.248,157.833
C04258=1038.845,212.440,-104.697,170.816,41.249,157.834
C04259=1038.851,212.688,-104.723,170.819,41.251,157.834
C04260=1038.858,212.936,-104.750,170.820,41.253,157.835
C04261=1038.864,213.185,-104.777,170.822,41.254,157.835
C04262=1038.871,213.433,-104.803,170.825,41.255,157.835
C04263=1038.878,213.682,-104.831,170.827,41.257,157.836
C04264=1038.885,213.931,-104.858,170.830,41.258,157.836
C04265=1038.890,214.179,-104.884,170.832,41.260,157.837
C04266=1038.897,214.427,-104.912,170.835,41.261,157.837
C04267=1038.904,214.676,-104.938,170.836,41.263,157.838
C04268=1038.910,214.924,-104.966,170.839,41.264,157.838
C04269=1038.917,215.173,-104.992,170.841,41.266,157.838
C04270=1038.924,215.422,-105.019,170.844,41.267,157.839
C04271=1038.931,215.670,-105.046,170.846,41.268,157.839
C04272=1038.937,215.918,-105.073,170.849,41.270,157.840
C04273=1038.944,216.166,-105.100,170.851,41.271,157.840
C04274=1038.951,216.415,-105.127,170.854,41.272,157.841
C04275=1038.958,216.664,-105.155,170.856,41.274,157.841
C04276=1038.964,216.912,-105.181,170.859,41.276,157.842
C04277=1038.970,217.161,-105.208,170.860,41.277,157.842
C04278=1038.978,217.409,-105.235,170.863,41.278,157.842
C04279=1038.984,217.658,-105.262,170.865,41.280,157.843
C04280=1038.991,217.905,-105.289,170.868,41.282,157.843
C04281=1038.997,218.155,-105.316,170.870,41.283,157.844
C04282=1039.005,218.403,-105.343,170.873,41.284,157.844
C04283=1039.012,218.651,-105.371,170.875,41.286,157.845
C04284=1039.017,218.899,-105.397,170.878,41.287,157.845
C04285=1039.025,219.148,-105.424,170.880,41.288,157.845
C04286=1039.031,219.397,-105.451,170.883,41.290,157.846
C04287=1039.038,219.645,-105.479,170.885,41.291,157.846
C04288=1039.045,219.894,-105.506,170.888,41.293,157.847
C04289=1039.053,220.213,-105.541,170.890,41.295,157.847
C04290=1039.062,220.533,-105.576,170.894,41.296,157.848
C04291=1039.070,220.854,-105.611,170.896,41.299,157.848
C04292=1039.079,221.174,-105.647,170.900,41.300,157.849
C04293=1039.085,221.421,-105.673,170.903,41.302,157.849
C04294=1039.092,221.670,-105.701,170.905,41.303,157.850
C04295=1039.099,221.918,-105.729,170.908,41.305,157.850
C04296=1039.105,222.167,-105.756,170.910,41.306,157.851
C04297=1039.112,222.416,-105.783,170.913,41.307,157.851
C04298=1039.118,222.663,-105.811,170.914,41.309,157.852
C04299=1039.125,222.912,-105.837,170.917,41.311,157.852
C04300=1039.132,223.161,-105.865,170.919,41.312,157.852
C04301=1039.138,223.409,-105.893,170.922,41.313,157.853
C04302=1039.145,223.658,-105.920,170.924,41.315,157.853
C04303=1039.152,223.906,-105.948,170.927,41.317,157.854
C04304=1039.158,224.155,-105.975,170.929,41.318,157.854
C04305=1039.164,224.403,-106.003,170.932,41.319,157.855
C04306=1039.172,224.651,-106.030,170.934,41.321,157.855
C04307=1039.178,224.899,-106.057,170.937,41.322,157.856
C04308=1039.185,225.148,-106.085,170.939,41.324,157.856
C04309=1039.192,225.396,-106.113,170.942,41.325,157.856
C04310=1039.198,225.645,-106.141,170.944,41.327,157.857
C04311=1039.205,225.894,-106.168,170.947,41.328,157.857
C04312=1039.211,226.142,-106.195,170.949,41.330,157.858
C04313=1039.219,226.390,-106.223,170.952,41.331,157.858
C04314=1039.225,226.638,-106.250,170.954,41.332,157.859
C04315=1039.232,226.886,-106.278,170.957,41.334,157.859
C04316=1039.238,227.135,-106.305,170.960,41.335,157.860
C04317=1039.245,227.383,-106.333,170.963,41.336,157.860
C04318=1039.252,227.632,-106.361,170.965,41.338,157.861
C04319=1039.258,227.880,-106.389,170.968,41.340,157.861
C04320=1039.265,228.129,-106.416,170.970,41.341,157.861
C04321=1039.272,228.377,-106.443,170.972,41.342,157.862
C04322=1039.278,228.626,-106.472,170.975,41.344,157.862
C04323=1039.285,228.874,-106.499,170.978,41.345,157.863
C04324=1039.292,229.122,-106.527,170.980,41.347,157.863
C04325=1039.298,229.371,-106.555,170.982,41.348,157.864
C04326=1039.305,229.619,-106.583,170.985,41.350,157.864
C04327=1039.312,229.868,-106.610,170.988,41.351,157.865
C04328=1039.319,230.116,-106.638,170.990,41.353,157.865
C04329=1039.325,230.365,-106.666,170.993,41.354,157.866
C04330=1039.332,230.613,-106.694,170.995,41.356,157.866
C04331=1039.339,230.861,-106.722,170.998,41.357,157.866
C04332=1039.346,231.109,-106.750,171.000,41.359,157.867
C04333=1039.351,231.358,-106.778,171.003,41.360,157.867
C04334=1039.358,231.607,-106.806,171.005,41.362,157.868
C04335=1039.365,231.855,-106.834,171.008,41.363,157.868
C04336=1039.372,232.103,-106.861,171.011,41.365,157.869
C04337=1039.379,232.351,-106.890,171.014,41.366,157.869
C04338=1039.385,232.599,-106.917,171.016,41.367,157.870
C04339=1039.391,232.848,-106.945,171.019,41.369,157.870
C04340=1039.397,233.096,-106.973,171.021,41.371,157.871
C04341=1039.404,233.344,-107.002,171.024,41.372,157.871
C04342=1039.411,233.592,-107.029,171.026,41.374,157.872
C04343=1039.417,233.842,-107.058,171.029,41.375,157.872
C04344=1039.424,234.090,-107.086,171.031,41.377,157.872
C04345=1039.433,234.402,-107.121,171.035,41.378,157.873
C04346=1039.441,234.715,-107.156,171.038,41.381,157.874
C04347=1039.449,235.027,-107.192,171.041,41.382,157.874
C04348=1039.458,235.339,-107.228,171.045,41.384,157.875
C04349=1039.464,235.588,-107.255,171.048,41.386,157.875
C04350=1039.470,235.837,-107.284,171.050,41.387,157.876
C04351=1039.477,236.084,-107.312,171.053,41.389,157.876
C04352=1039.484,236.333,-107.340,171.055,41.390,157.877
C04353=1039.491,236.581,-107.368,171.058,41.392,157.877
C04354=1039.497,236.829,-107.397,171.061,41.393,157.878
C04355=1039.504,237.079,-107.425,171.064,41.395,157.878
C04356=1039.511,237.326,-107.453,171.066,41.396,157.879
C04357=1039.518,237.575,-107.481,171.069,41.398,157.879
C04358=1039.524,237.823,-107.510,171.071,41.399,157.879
C04359=1039.531,238.071,-107.538,171.074,41.400,157.880
C04360=1039.538,238.319,-107.566,171.076,41.402,157.880
C04361=1039.544,238.568,-107.594,171.080,41.403,157.881
C04362=1039.551,238.816,-107.623,171.082,41.405,157.881
C04363=1039.558,239.065,-107.651,171.085,41.407,157.882
C04364=1039.564,239.313,-107.680,171.087,41.408,157.882
C04365=1039.571,239.561,-107.708,171.090,41.410,157.883
C04366=1039.578,239.809,-107.736,171.093,41.411,157.883
C04367=1039.584,240.058,-107.764,171.096,41.412,157.884
C04368=1039.591,240.306,-107.793,171.098,41.414,157.884
C04369=1039.598,240.554,-107.821,171.101,41.415,157.885
C04370=1039.604,240.803,-107.850,171.104,41.417,157.885
C04371=1039.611,241.051,-107.878,171.106,41.419,157.886
C04372=1039.617,241.299,-107.907,171.110,41.420,157.886
C04373=1039.624,241.548,-107.935,171.112,41.422,157.887
C04374=1039.630,241.796,-107.964,171.115,41.423,157.887
C04375=1039.637,242.044,-107.993,171.117,41.425,157.888
C04376=1039.643,242.292,-108.021,171.120,41.426,157.888
C04377=1039.650,242.541,-108.050,171.122,41.428,157.888
C04378=1039.657,242.789,-108.079,171.126,41.429,157.889
C04379=1039.663,243.037,-108.108,171.129,41.431,157.889
C04380=1039.670,243.285,-108.136,171.131,41.433,157.890
C04381=1039.676,243.534,-108.165,171.134,41.434,157.890
C04382=1039.683,243.782,-108.194,171.136,41.436,157.891
C04383=1039.690,244.030,-108.223,171.140,41.437,157.891
C04384=1039.696,244.279,-108.251,171.142,41.439,157.892
C04385=1039.703,244.527,-108.279,171.145,41.440,157.892
C04386=1039.709,244.775,-108.308,171.147,41.442,157.893
C04387=1039.716,245.024,-108.338,171.151,41.443,157.893
C04388=1039.723,245.272,-108.366,171.153,41.445,157.894
C04389=1039.729,245.520,-108.395,171.156,41.447,157.894
C04390=1039.736,245.768,-108.424,171.159,41.448,157.895
C04391=1039.742,246.016,-108.453,171.161,41.450,157.895
C04392=1039.749,246.265,-108.483,171.165,41.451,157.896
C04393=1039.756,246.513,-108.511,171.167,41.453,157.896
C04394=1039.762,246.761,-108.540,171.170,41.454,157.897
C04395=1039.768,247.009,-108.569,171.172,41.456,157.897
C04396=1039.775,247.257,-108.598,171.175,41.458,157.898
C04397=1039.781,247.506,-108.628,171.179,41.460,157.898
C04398=1039.788,247.754,-108.657,171.181,41.461,157.899
C04399=1039.794,248.002,-108.686,171.184,41.463,157.899
C04400=1039.801,248.250,-108.714,171.186,41.464,157.900
C04401=1039.809,248.558,-108.750,171.190,41.466,157.901
C04402=1039.817,248.864,-108.786,171.194,41.468,157.901
C04403=1039.825,249.170,-108.822,171.197,41.470,157.902
C04404=1039.834,249.477,-108.858,171.201,41.472,157.902
C04405=1039.840,249.725,-108.887,171.204,41.474,157.903
C04406=1039.846,249.974,-108.916,171.206,41.475,157.903
C04407=1039.853,250.222,-108.946,171.209,41.477,157.904
C04408=1039.859,250.471,-108.975,171.212,41.478,157.904
C04409=1039.866,250.718,-109.005,171.215,41.480,157.905
C04410=1039.872,250.966,-109.034,171.218,41.482,157.905
C04411=1039.879,251.215,-109.063,171.221,41.483,157.906
C04412=1039.886,251.463,-109.091,171.224,41.485,157.906
C04413=1039.892,251.711,-109.120,171.226,41.487,157.907
C04414=1039.899,251.960,-109.150,171.229,41.488,157.907
C04415=1039.906,252.207,-109.180,171.232,41.490,157.908
C04416=1039.912,252.456,-109.209,171.235,41.491,157.908
C04417=1039.919,252.704,-109.238,171.237,41.493,157.909
C04418=1039.925,252.952,-109.267,171.241,41.494,157.909
C04419=1039.932,253.201,-109.297,171.244,41.496,157.910
C04420=1039.939,253.448,-109.326,171.246,41.498,157.911
C04421=1039.945,253.697,-109.355,171.250,41.499,157.911
C04422=1039.952,253.945,-109.385,171.252,41.501,157.912
C04423=1039.959,254.193,-109.414,171.255,41.503,157.912
C04424=1039.966,254.442,-109.443,171.259,41.504,157.913
C04425=1039.972,254.689,-109.473,171.261,41.506,157.913
C04426=1039.979,254.938,-109.502,171.264,41.507,157.914
C04427=1039.985,255.186,-109.532,171.267,41.509,157.914
C04428=1039.992,255.434,-109.561,171.270,41.510,157.915
C04429=1039.999,255.683,-109.591,171.273,41.512,157.915
C04430=1040.006,255.930,-109.619,171.276,41.513,157.916
C04431=1040.013,256.179,-109.649,171.279,41.515,157.916
C04432=1040.019,256.427,-109.678,171.282,41.517,157.917
C04433=1040.026,256.675,-109.708,171.285,41.518,157.917
C04434=1040.032,256.923,-109.737,171.287,41.520,157.918
C04435=1040.040,257.171,-109.768,171.291,41.521,157.918
C04436=1040.046,257.419,-109.797,171.293,41.523,157.919
C04437=1040.053,257.668,-109.826,171.297,41.524,157.919
C04438=1040.059,257.916,-109.856,171.300,41.526,157.920
C04439=1040.066,258.165,-109.885,171.302,41.528,157.920
C04440=1040.073,258.412,-109.915,171.306,41.530,157.921
C04441=1040.080,258.661,-109.944,171.308,41.531,157.921
C04442=1040.087,258.908,-109.974,171.312,41.533,157.922
C04443=1040.094,259.157,-110.003,171.315,41.534,157.922
C04444=1040.100,259.404,-110.033,171.318,41.536,157.923
C04445=1040.107,259.653,-110.063,171.321,41.537,157.923
C04446=1040.114,259.902,-110.092,171.323,41.539,157.924
C04447=1040.121,260.149,-110.122,171.327,41.540,157.924
C04448=1040.128,260.398,-110.151,171.329,41.542,157.925
C04449=1040.134,260.645,-110.181,171.333,41.544,157.925
C04450=1040.141,260.894,-110.211,171.336,41.545,157.926
C04451=1040.148,261.142,-110.241,171.339,41.547,157.926
C04452=1040.155,261.390,-110.270,171.342,41.548,157.927
C04453=1040.162,261.638,-110.301,171.345,41.550,157.928
C04454=1040.168,261.886,-110.330,171.348,41.551,157.928
C04455=1040.175,262.135,-110.360,171.350,41.553,157.928
C04456=1040.182,262.382,-110.389,171.354,41.555,157.929
C04457=1040.190,262.688,-110.426,171.358,41.557,157.930
C04458=1040.198,262.994,-110.463,171.362,41.559,157.930
C04459=1040.206,263.298,-110.500,171.365,41.561,157.931
C04460=1040.215,263.603,-110.537,171.369,41.563,157.932
C04461=1040.221,263.852,-110.567,171.372,41.565,157.932
C04462=1040.228,264.099,-110.597,171.375,41.566,157.933
C04463=1040.235,264.348,-110.627,171.378,41.568,157.933
C04464=1040.241,264.596,-110.658,171.382,41.570,157.934
C04465=1040.248,264.844,-110.688,171.384,41.571,157.934
C04466=1040.255,265.092,-110.718,171.388,41.573,157.935
C04467=1040.261,265.340,-110.748,171.390,41.575,157.936
C04468=1040.268,265.588,-110.778,171.394,41.576,157.936
C04469=1040.275,265.836,-110.808,171.397,41.579,157.937
C04470=1040.281,266.085,-110.838,171.400,41.580,157.937
C04471=1040.288,266.333,-110.868,171.403,41.582,157.938
C04472=1040.295,266.581,-110.898,171.407,41.584,157.938
C04473=1040.301,266.829,-110.929,171.409,41.585,157.939
C04474=1040.308,267.077,-110.959,171.413,41.587,157.939
C04475=1040.315,267.325,-110.990,171.416,41.589,157.940
C04476=1040.321,267.572,-111.020,171.419,41.590,157.941
C04477=1040.328,267.821,-111.050,171.422,41.592,157.941
C04478=1040.335,268.069,-111.081,171.425,41.594,157.942
C04479=1040.341,268.317,-111.111,171.428,41.595,157.942
C04480=1040.348,268.565,-111.141,171.432,41.597,157.943
C04481=1040.355,268.813,-111.171,171.434,41.599,157.943
C04482=1040.361,269.061,-111.201,171.438,41.600,157.944
C04483=1040.368,269.309,-111.233,171.441,41.603,157.945
C04484=1040.375,269.557,-111.263,171.444,41.604,157.945
C04485=1040.382,269.806,-111.293,171.447,41.606,157.946
C04486=1040.388,270.053,-111.323,171.451,41.608,157.946
C04487=1040.395,270.302,-111.354,171.453,41.609,157.947
C04488=1040.402,270.549,-111.385,171.457,41.611,157.947
C04489=1040.409,270.798,-111.416,171.460,41.613,157.948
C04490=1040.415,271.045,-111.445,171.463,41.615,157.949
C04491=1040.421,271.294,-111.476,171.467,41.616,157.949
C04492=1040.429,271.541,-111.507,171.469,41.618,157.950
C04493=1040.435,271.790,-111.538,171.473,41.620,157.950
C04494=1040.441,272.038,-111.568,171.476,41.621,157.951
C04495=1040.449,272.285,-111.599,171.479,41.623,157.951
C04496=1040.455,272.534,-111.629,171.482,41.625,157.952
C04497=1040.461,272.782,-111.660,171.486,41.627,157.953
C04498=1040.468,273.029,-111.691,171.489,41.628,157.953
C04499=1040.475,273.278,-111.721,171.492,41.631,157.954
C04500=1040.481,273.526,-111.753,171.496,41.632,157.954
C04501=1040.489,273.774,-111.783,171.498,41.634,157.955
C04502=1040.495,274.022,-111.814,171.502,41.636,157.955
C04503=1040.501,274.270,-111.845,171.505,41.638,157.956
C04504=1040.508,274.518,-111.875,171.508,41.639,157.957
C04505=1040.515,274.766,-111.906,171.512,41.641,157.957
C04506=1040.522,275.014,-111.938,171.515,41.643,157.958
C04507=1040.529,275.262,-111.968,171.518,41.645,157.958
C04508=1040.535,275.509,-111.999,171.521,41.647,157.959
C04509=1040.541,275.758,-112.030,171.525,41.648,157.960
C04510=1040.548,276.006,-112.061,171.528,41.650,157.960
C04511=1040.555,276.254,-112.091,171.531,41.652,157.961
C04512=1040.562,276.502,-112.123,171.535,41.654,157.961
C04513=1040.570,276.812,-112.162,171.538,41.656,157.962
C04514=1040.579,277.121,-112.200,171.543,41.658,157.963
C04515=1040.587,277.431,-112.239,171.547,41.660,157.964
C04516=1040.595,277.741,-112.277,171.551,41.663,157.964
C04517=1040.603,277.989,-112.308,171.555,41.664,157.965
C04518=1040.609,278.237,-112.340,171.557,41.667,157.965
C04519=1040.616,278.485,-112.370,171.561,41.668,157.966
C04520=1040.622,278.733,-112.401,171.565,41.670,157.967
C04521=1040.629,278.980,-112.433,171.568,41.672,157.967
C04522=1040.635,279.228,-112.464,171.571,41.674,157.968
C04523=1040.642,279.476,-112.496,171.575,41.676,157.968
C04524=1040.649,279.725,-112.526,171.578,41.678,157.969
C04525=1040.655,279.973,-112.558,171.581,41.680,157.970
C04526=1040.662,280.221,-112.589,171.585,41.681,157.970
C04527=1040.669,280.469,-112.621,171.588,41.683,157.971
C04528=1040.675,280.716,-112.652,171.591,41.685,157.972
C04529=1040.683,280.964,-112.683,171.595,41.687,157.972
C04530=1040.690,281.212,-112.714,171.598,41.689,157.973
C04531=1040.696,281.460,-112.746,171.602,41.691,157.973
C04532=1040.703,281.708,-112.777,171.605,41.693,157.974
C04533=1040.710,281.956,-112.808,171.608,41.695,157.975
C04534=1040.716,282.204,-112.839,171.612,41.697,157.975
C04535=1040.722,282.451,-112.870,171.615,41.699,157.976
C04536=1040.729,282.699,-112.902,171.618,41.700,157.976
C04537=1040.736,282.947,-112.933,171.622,41.702,157.977
C04538=1040.743,283.195,-112.965,171.625,41.704,157.978
C04539=1040.750,283.444,-112.997,171.629,41.706,157.978
C04540=1040.757,283.692,-113.028,171.632,41.708,157.979
C04541=1040.764,283.939,-113.060,171.636,41.710,157.980
C04542=1040.770,284.187,-113.092,171.639,41.712,157.980
C04543=1040.776,284.435,-113.124,171.642,41.714,157.981
C04544=1040.783,284.683,-113.155,171.646,41.715,157.981
C04545=1040.790,284.931,-113.186,171.649,41.717,157.982
C04546=1040.797,285.179,-113.218,171.653,41.719,157.983
C04547=1040.803,285.427,-113.249,171.656,41.721,157.983
C04548=1040.810,285.674,-113.281,171.660,41.723,157.984
C04549=1040.817,285.922,-113.312,171.663,41.725,157.985
C04550=1040.824,286.170,-113.344,171.667,41.727,157.985
C04551=1040.830,286.418,-113.376,171.671,41.729,157.986
C04552=1040.837,286.665,-113.407,171.674,41.731,157.987
C04553=1040.844,286.914,-113.439,171.677,41.733,157.987
C04554=1040.851,287.162,-113.470,171.681,41.734,157.988
C04555=1040.858,287.409,-113.503,171.685,41.736,157.989
C04556=1040.865,287.657,-113.534,171.687,41.739,157.989
C04557=1040.871,287.905,-113.566,171.691,41.741,157.990
C04558=1040.878,288.153,-113.598,171.695,41.743,157.991
C04559=1040.885,288.401,-113.630,171.699,41.745,157.991
C04560=1040.891,288.648,-113.661,171.702,41.747,157.992
C04561=1040.899,288.896,-113.694,171.705,41.749,157.992
C04562=1040.905,289.145,-113.726,171.709,41.751,157.993
C04563=1040.912,289.392,-113.758,171.713,41.753,157.994
C04564=1040.919,289.640,-113.789,171.717,41.755,157.995
C04565=1040.926,289.888,-113.821,171.719,41.756,157.995
C04566=1040.932,290.135,-113.853,171.723,41.758,157.996
C04567=1040.939,290.384,-113.885,171.727,41.760,157.996
C04568=1040.946,290.631,-113.917,171.730,41.762,157.997
C04569=1040.955,290.952,-113.959,171.736,41.765,157.998
C04570=1040.963,291.275,-114.001,171.740,41.768,157.999
C04571=1040.972,291.596,-114.042,171.745,41.770,158.000
C04572=1040.981,291.918,-114.085,171.749,41.773,158.001
C04573=1040.988,292.166,-114.116,171.752,41.775,158.001
C04574=1040.995,292.413,-114.148,171.756,41.777,158.002
C04575=1041.001,292.661,-114.180,171.760,41.779,158.003
C04576=1041.008,292.909,-114.212,171.764,41.781,158.003
C04577=1041.015,293.157,-114.245,171.767,41.783,158.004
C04578=1041.021,293.405,-114.277,171.771,41.785,158.005
C04579=1041.028,293.652,-114.309,171.775,41.787,158.005
C04580=1041.035,293.900,-114.342,171.778,41.789,158.006
C04581=1041.042,294.148,-114.374,171.782,41.792,158.007
C04582=1041.049,294.396,-114.406,171.785,41.794,158.007
C04583=1041.055,294.643,-114.438,171.789,41.796,158.008
C04584=1041.063,294.891,-114.471,171.793,41.798,158.009
C04585=1041.069,295.139,-114.504,171.797,41.800,158.009
C04586=1041.076,295.387,-114.535,171.800,41.802,158.010
C04587=1041.083,295.635,-114.568,171.804,41.804,158.011
C04588=1041.089,295.883,-114.601,171.807,41.807,158.012
C04589=1041.096,296.130,-114.633,171.811,41.809,158.012
C04590=1041.103,296.377,-114.666,171.815,41.811,158.013
C04591=1041.109,296.626,-114.699,171.818,41.813,158.014
C04592=1041.116,296.873,-114.732,171.822,41.815,158.014
C04593=1041.123,297.121,-114.764,171.826,41.817,158.015
C04594=1041.129,297.368,-114.797,171.830,41.819,158.016
C04595=1041.136,297.616,-114.830,171.834,41.822,158.017
C04596=1041.142,297.864,-114.862,171.837,41.824,158.017
C04597=1041.149,298.112,-114.895,171.841,41.826,158.018
C04598=1041.156,298.360,-114.928,171.844,41.828,158.019
C04599=1041.162,298.607,-114.960,171.848,41.830,158.019
C04600=1041.169,298.855,-114.993,171.852,41.832,158.020
C04601=1041.176,299.103,-115.026,171.856,41.834,158.021
C04602=1041.183,299.350,-115.058,171.860,41.837,158.022
C04603=1041.189,299.597,-115.092,171.864,41.839,158.022
C04604=1041.196,299.846,-115.125,171.867,41.841,158.023
C04605=1041.202,300.093,-115.158,171.871,41.844,158.024
C04606=1041.209,300.342,-115.191,171.875,41.845,158.024
C04607=1041.216,300.589,-115.223,171.879,41.847,158.025
C04608=1041.223,300.836,-115.257,171.883,41.850,158.026
C04609=1041.230,301.084,-115.290,171.886,41.852,158.027
C04610=1041.236,301.332,-115.322,171.890,41.855,158.027
C04611=1041.243,301.580,-115.355,171.893,41.857,158.028
C04612=1041.250,301.827,-115.388,171.897,41.859,158.029
C04613=1041.257,302.075,-115.421,171.901,41.861,158.030
C04614=1041.264,302.322,-115.454,171.905,41.863,158.030
C04615=1041.270,302.571,-115.487,171.909,41.866,158.031
C04616=1041.277,302.818,-115.521,171.913,41.868,158.032
C04617=1041.285,303.066,-115.553,171.916,41.870,158.032
C04618=1041.291,303.313,-115.586,171.920,41.872,158.033
C04619=1041.298,303.561,-115.620,171.924,41.874,158.034
C04620=1041.305,303.809,-115.653,171.928,41.877,158.035
C04621=1041.312,304.056,-115.686,171.932,41.879,158.035
C04622=1041.318,304.304,-115.719,171.936,41.882,158.036
C04623=1041.326,304.552,-115.752,171.940,41.884,158.037
C04624=1041.332,304.799,-115.785,171.944,41.886,158.038
C04625=1041.341,305.137,-115.831,171.950,41.889,158.039
C04626=1041.351,305.476,-115.876,171.955,41.892,158.040
C04627=1041.360,305.814,-115.921,171.960,41.895,158.041
C04628=1041.370,306.152,-115.966,171.965,41.898,158.042
C04629=1041.377,306.400,-116.000,171.969,41.901,158.043
C04630=1041.384,306.647,-116.033,171.973,41.903,158.043
C04631=1041.391,306.895,-116.066,171.977,41.905,158.044
C04632=1041.398,307.143,-116.100,171.981,41.907,158.045
C04633=1041.404,307.390,-116.133,171.985,41.910,158.046
C04634=1041.412,307.637,-116.166,171.990,41.912,158.046
C04635=1041.419,307.885,-116.200,171.993,41.914,158.047
C04636=1041.426,308.133,-116.233,171.997,41.916,158.048
C04637=1041.433,308.380,-116.267,172.001,41.919,158.049
C04638=1041.440,308.628,-116.300,172.005,41.921,158.049
C04639=1041.446,308.876,-116.333,172.009,41.923,158.050
C04640=1041.453,309.123,-116.367,172.013,41.926,158.051
C04641=1041.461,309.371,-116.400,172.017,41.928,158.052
C04642=1041.469,309.618,-116.434,172.021,41.930,158.053
C04643=1041.475,309.866,-116.467,172.026,41.932,158.053
C04644=1041.482,310.114,-116.501,172.030,41.935,158.054
C04645=1041.489,310.361,-116.534,172.033,41.937,158.055
C04646=1041.496,310.609,-116.568,172.037,41.939,158.056
C04647=1041.503,310.857,-116.601,172.041,41.942,158.056
C04648=1041.510,311.104,-116.635,172.045,41.944,158.057
C04649=1041.518,311.352,-116.668,172.049,41.946,158.058
C04650=1041.525,311.599,-116.702,172.054,41.949,158.059
C04651=1041.532,311.847,-116.736,172.058,41.951,158.060
C04652=1041.539,312.094,-116.769,172.062,41.953,158.060
C04653=1041.546,312.342,-116.803,172.066,41.956,158.061
C04654=1041.553,312.590,-116.837,172.070,41.958,158.062
C04655=1041.560,312.837,-116.871,172.074,41.961,158.063
C04656=1041.566,313.084,-116.905,172.079,41.963,158.064
C04657=1041.573,313.332,-116.939,172.083,41.966,158.065
C04658=1041.580,313.580,-116.973,172.086,41.968,158.065
C04659=1041.587,313.827,-117.008,172.090,41.971,158.066
C04660=1041.593,314.074,-117.042,172.094,41.973,158.067
C04661=1041.600,314.322,-117.076,172.098,41.976,158.068
C04662=1041.607,314.570,-117.110,172.102,41.978,158.069
C04663=1041.614,314.818,-117.144,172.107,41.981,158.069
C04664=1041.621,315.065,-117.179,172.111,41.983,158.070
C04665=1041.627,315.312,-117.213,172.115,41.986,158.071
C04666=1041.634,315.560,-117.247,172.119,41.988,158.072
C04667=1041.641,315.808,-117.281,172.123,41.991,158.073
C04668=1041.648,316.055,-117.316,172.127,41.993,158.074
C04669=1041.655,316.303,-117.349,172.132,41.996,158.074
C04670=1041.662,316.551,-117.384,172.136,41.998,158.075
C04671=1041.669,316.798,-117.418,172.140,42.001,158.076
C04672=1041.675,317.045,-117.452,172.144,42.004,158.077
C04673=1041.682,317.293,-117.486,172.148,42.007,158.078
C04674=1041.689,317.540,-117.521,172.153,42.009,158.079
C04675=1041.696,317.788,-117.555,172.157,42.012,158.080
C04676=1041.703,318.035,-117.590,172.161,42.014,158.081
C04677=1041.710,318.283,-117.624,172.165,42.017,158.081
C04678=1041.717,318.530,-117.659,172.170,42.019,158.082
C04679=1041.724,318.778,-117.693,172.174,42.022,158.083
C04680=1041.731,319.025,-117.728,172.178,42.024,158.084
C04681=1041.741,319.368,-117.776,172.185,42.028,158.085
C04682=1041.751,319.711,-117.824,172.190,42.032,158.086
C04683=1041.760,320.054,-117.871,172.197,42.035,158.088
C04684=1041.769,320.396,-117.919,172.202,42.039,158.089
C04685=1041.777,320.644,-117.955,172.206,42.041,158.090
C04686=1041.784,320.892,-117.988,172.211,42.044,158.090
C04687=1041.791,321.139,-118.024,172.215,42.046,158.091
C04688=1041.798,321.387,-118.057,172.219,42.049,158.092
C04689=1041.805,321.634,-118.093,172.224,42.052,158.093
C04690=1041.812,321.881,-118.127,172.228,42.054,158.094
C04691=1041.819,322.129,-118.162,172.232,42.057,158.095
C04692=1041.826,322.377,-118.196,172.237,42.060,158.096
C04693=1041.833,322.624,-118.231,172.241,42.062,158.097
C04694=1041.841,322.871,-118.266,172.245,42.065,158.098
C04695=1041.848,323.120,-118.301,172.250,42.067,158.098
C04696=1041.855,323.367,-118.335,172.255,42.071,158.099
C04697=1041.862,323.614,-118.370,172.259,42.073,158.100
C04698=1041.869,323.861,-118.405,172.264,42.075,158.101
C04699=1041.876,324.108,-118.440,172.268,42.078,158.102
C04700=1041.883,324.356,-118.475,172.272,42.081,158.103
C04701=1041.891,324.604,-118.509,172.277,42.084,158.104
C04702=1041.897,324.852,-118.544,172.281,42.086,158.105
C04703=1041.905,325.099,-118.579,172.285,42.089,158.106
C04704=1041.912,325.346,-118.614,172.290,42.092,158.107
C04705=1041.920,325.594,-118.649,172.294,42.095,158.108
C04706=1041.927,325.841,-118.684,172.299,42.097,158.108
C04707=1041.933,326.088,-118.719,172.303,42.100,158.109
C04708=1041.941,326.336,-118.754,172.307,42.103,158.110
C04709=1041.948,326.584,-118.789,172.312,42.105,158.111
C04710=1041.956,326.831,-118.824,172.316,42.108,158.112
C04711=1041.963,327.078,-118.859,172.321,42.111,158.113
C04712=1041.970,327.326,-118.894,172.325,42.113,158.114
C04713=1041.977,327.573,-118.929,172.330,42.116,158.115
C04714=1041.984,327.820,-118.964,172.335,42.119,158.116
C04715=1041.992,328.068,-118.999,172.339,42.122,158.117
C04716=1041.999,328.316,-119.034,172.344,42.124,158.118
C04717=1042.007,328.563,-119.070,172.348,42.127,158.119
C04718=1042.014,328.810,-119.105,172.353,42.130,158.119
C04719=1042.021,329.057,-119.140,172.357,42.133,158.120
C04720=1042.028,329.306,-119.176,172.362,42.135,158.121
C04721=1042.035,329.552,-119.211,172.366,42.138,158.122
C04722=1042.042,329.800,-119.247,172.372,42.141,158.123
C04723=1042.050,330.048,-119.282,172.376,42.144,158.124
C04724=1042.057,330.294,-119.318,172.380,42.147,158.125
C04725=1042.063,330.542,-119.353,172.385,42.150,158.126
C04726=1042.071,330.790,-119.388,172.389,42.153,158.127
C04727=1042.078,331.037,-119.424,172.395,42.156,158.128
C04728=1042.085,331.285,-119.460,172.399,42.158,158.129
C04729=1042.092,331.531,-119.496,172.404,42.161,158.130
C04730=1042.099,331.779,-119.531,172.408,42.164,158.131
C04731=1042.107,332.026,-119.567,172.413,42.167,158.132
C04732=1042.114,332.274,-119.602,172.417,42.170,158.133
C04733=1042.121,332.521,-119.638,172.422,42.173,158.134
C04734=1042.128,332.768,-119.674,172.427,42.176,158.135
C04735=1042.136,333.016,-119.710,172.432,42.179,158.136
C04736=1042.143,333.263,-119.746,172.436,42.182,158.137
C04737=1042.155,333.670,-119.805,172.444,42.187,158.139
C04738=1042.167,334.078,-119.864,172.452,42.192,158.140
C04739=1042.179,334.486,-119.923,172.460,42.197,158.142
C04740=1042.191,334.893,-119.981,172.468,42.202,158.144
C04741=1042.198,335.140,-120.017,172.472,42.205,158.145
C04742=1042.205,335.388,-120.054,172.477,42.208,158.146
C04743=1042.213,335.635,-120.090,172.481,42.211,158.147
C04744=1042.220,335.882,-120.126,172.487,42.214,158.148
C04745=1042.227,336.130,-120.161,172.491,42.217,158.149
C04746=1042.234,336.377,-120.198,172.496,42.220,158.150
C04747=1042.241,336.625,-120.234,172.500,42.223,158.151
C04748=1042.248,336.871,-120.270,172.506,42.226,158.152
C04749=1042.256,337.119,-120.306,172.511,42.229,158.153
C04750=1042.263,337.367,-120.343,172.515,42.232,158.154
C04751=1042.270,337.613,-120.379,172.520,42.235,158.155
C04752=1042.278,337.861,-120.415,172.525,42.238,158.156
C04753=1042.284,338.108,-120.451,172.530,42.241,158.157
C04754=1042.292,338.355,-120.487,172.535,42.244,158.158
C04755=1042.300,338.603,-120.524,172.539,42.247,158.159
C04756=1042.307,338.849,-120.559,172.545,42.251,158.160
C04757=1042.314,339.097,-120.596,172.549,42.254,158.161
C04758=1042.322,339.344,-120.633,172.554,42.257,158.162
C04759=1042.329,339.591,-120.669,172.559,42.260,158.163
C04760=1042.336,339.838,-120.706,172.564,42.264,158.164
C04761=1042.342,340.051,-120.737,172.569,42.266,158.165
C04762=1042.348,340.263,-120.768,172.573,42.268,158.166
C04763=1042.355,340.476,-120.800,172.577,42.271,158.167
C04764=1042.362,340.689,-120.831,172.581,42.274,158.168
C04765=1042.368,340.901,-120.862,172.585,42.277,158.169
C04766=1042.374,341.114,-120.894,172.589,42.280,158.170
C04767=1042.380,341.326,-120.925,172.594,42.282,158.171
C04768=1042.387,341.539,-120.956,172.598,42.285,158.172
C04769=1042.395,341.786,-120.993,172.603,42.288,158.173
C04770=1042.401,342.033,-121.030,172.608,42.292,158.174
C04771=1042.409,342.280,-121.066,172.613,42.294,158.175
C04772=1042.416,342.527,-121.104,172.618,42.298,158.176
C04773=1042.424,342.775,-121.140,172.623,42.301,158.177
C04774=1042.431,343.022,-121.177,172.628,42.305,158.178
C04775=1042.438,343.269,-121.213,172.634,42.308,158.179
C04776=1042.445,343.516,-121.251,172.638,42.311,158.181
C04777=1042.453,343.763,-121.287,172.643,42.314,158.182
C04778=1042.460,344.010,-121.324,172.649,42.318,158.183
C04779=1042.467,344.258,-121.361,172.653,42.321,158.184
C04780=1042.475,344.505,-121.398,172.658,42.324,158.185
C04781=1042.482,344.752,-121.436,172.664,42.328,158.186
C04782=1042.490,344.999,-121.472,172.669,42.331,158.187
C04783=1042.497,345.246,-121.509,172.673,42.334,158.188
C04784=1042.505,345.493,-121.546,172.679,42.338,158.190
C04785=1042.512,345.741,-121.583,172.684,42.341,158.191
C04786=1042.519,345.988,-121.620,172.690,42.344,158.192
C04787=1042.527,346.235,-121.657,172.695,42.348,158.193
C04788=1042.534,346.482,-121.694,172.699,42.351,158.194
C04789=1042.541,346.730,-121.732,172.705,42.354,158.195
C04790=1042.549,346.976,-121.769,172.710,42.358,158.196
C04791=1042.556,347.223,-121.806,172.716,42.361,158.198
C04792=1042.564,347.471,-121.844,172.721,42.365,158.199
C04793=1042.574,347.806,-121.894,172.728,42.369,158.200
C04794=1042.584,348.139,-121.944,172.735,42.374,158.202
C04795=1042.594,348.474,-121.995,172.742,42.379,158.204
C04796=1042.604,348.808,-122.045,172.749,42.383,158.205
C04797=1042.611,349.055,-122.082,172.754,42.387,158.206
C04798=1042.619,349.302,-122.119,172.759,42.390,158.207
C04799=1042.627,349.550,-122.157,172.765,42.394,158.209
C04800=1042.635,349.796,-122.195,172.770,42.397,158.210
C04801=1042.643,350.043,-122.232,172.776,42.401,158.211
C04802=1042.650,350.290,-122.270,172.780,42.404,158.212
C04803=1042.657,350.538,-122.307,172.786,42.408,158.213
C04804=1042.664,350.785,-122.345,172.791,42.411,158.215
C04805=1042.672,351.032,-122.382,172.797,42.415,158.216
C04806=1042.679,351.278,-122.421,172.802,42.418,158.217
C04807=1042.687,351.526,-122.458,172.808,42.422,158.218
C04808=1042.694,351.773,-122.496,172.813,42.425,158.219
C04809=1042.702,352.020,-122.533,172.819,42.429,158.221
C04810=1042.710,352.267,-122.571,172.824,42.433,158.222
C04811=1042.717,352.514,-122.609,172.829,42.437,158.223
C04812=1042.725,352.760,-122.647,172.834,42.440,158.224
C04813=1042.732,353.008,-122.685,172.839,42.443,158.226
C04814=1042.740,353.255,-122.722,172.845,42.448,158.227
C04815=1042.747,353.502,-122.761,172.851,42.451,158.228
C04816=1042.754,353.749,-122.798,172.856,42.454,158.229
C04817=1042.763,353.996,-122.837,172.862,42.459,158.231
C04818=1042.770,354.243,-122.874,172.867,42.462,158.232
C04819=1042.777,354.490,-122.912,172.873,42.465,158.233
C04820=1042.785,354.737,-122.950,172.878,42.470,158.234
C04821=1042.793,354.984,-122.989,172.884,42.473,158.236
C04822=1042.800,355.231,-123.026,172.889,42.476,158.237
C04823=1042.808,355.478,-123.064,172.895,42.481,158.238
C04824=1042.817,355.725,-123.102,172.900,42.484,158.239
C04825=1042.824,355.972,-123.140,172.906,42.488,158.241
C04826=1042.832,356.219,-123.179,172.911,42.491,158.242
C04827=1042.839,356.466,-123.217,172.917,42.496,158.243
C04828=1042.847,356.713,-123.254,172.923,42.499,158.245
C04829=1042.854,356.960,-123.294,172.928,42.503,158.246
C04830=1042.862,357.207,-123.332,172.934,42.506,158.247
C04831=1042.869,357.453,-123.370,172.939,42.511,158.248
C04832=1042.877,357.700,-123.409,172.945,42.514,158.250
C04833=1042.885,357.947,-123.447,172.950,42.518,158.251
C04834=1042.893,358.194,-123.485,172.956,42.522,158.252
C04835=1042.900,358.441,-123.523,172.963,42.525,158.254
C04836=1042.908,358.689,-123.562,172.968,42.529,158.255
C04837=1042.915,358.935,-123.600,172.974,42.533,158.256
C04838=1042.923,359.183,-123.639,172.980,42.537,158.258
C04839=1042.931,359.429,-123.677,172.985,42.541,158.259
C04840=1042.939,359.676,-123.716,172.991,42.545,158.260
C04841=1042.947,359.922,-123.755,172.996,42.549,158.262
C04842=1042.955,360.169,-123.793,173.002,42.553,158.263
C04843=1042.962,360.416,-123.832,173.008,42.557,158.264
C04844=1042.970,360.664,-123.871,173.013,42.560,158.266
C04845=1042.978,360.910,-123.909,173.020,42.564,158.267
C04846=1042.986,361.157,-123.948,173.026,42.568,158.268
C04847=1042.993,361.403,-123.987,173.031,42.572,158.270
C04848=1043.001,361.651,-124.026,173.037,42.576,158.271
C04849=1043.012,361.991,-124.079,173.045,42.582,158.273
C04850=1043.023,362.331,-124.132,173.054,42.587,158.275
C04851=1043.033,362.672,-124.186,173.061,42.593,158.277
C04852=1043.045,363.011,-124.240,173.069,42.598,158.279
C04853=1043.051,363.258,-124.279,173.075,42.603,158.280
C04854=1043.060,363.505,-124.318,173.081,42.607,158.282
C04855=1043.067,363.752,-124.358,173.088,42.611,158.283
C04856=1043.075,363.998,-124.397,173.093,42.615,158.284
C04857=1043.082,364.246,-124.436,173.099,42.619,158.286
C04858=1043.091,364.492,-124.475,173.105,42.623,158.287
C04859=1043.098,364.739,-124.514,173.112,42.627,158.289
C04860=1043.106,364.986,-124.553,173.117,42.631,158.290
C04861=1043.114,365.232,-124.593,173.123,42.636,158.292
C04862=1043.121,365.479,-124.631,173.129,42.640,158.293
C04863=1043.129,365.726,-124.671,173.136,42.644,158.294
C04864=1043.138,365.972,-124.711,173.141,42.648,158.296
C04865=1043.145,366.219,-124.751,173.147,42.652,158.297
C04866=1043.154,366.467,-124.789,173.153,42.656,158.299
C04867=1043.161,366.713,-124.829,173.160,42.661,158.300
C04868=1043.169,366.959,-124.868,173.165,42.665,158.302
C04869=1043.177,367.206,-124.908,173.171,42.669,158.303
C04870=1043.185,367.453,-124.947,173.178,42.673,158.305
C04871=1043.193,367.700,-124.987,173.184,42.678,158.306
C04872=1043.201,367.947,-125.026,173.190,42.682,158.307
C04873=1043.208,368.193,-125.065,173.197,42.686,158.309
C04874=1043.217,368.440,-125.105,173.202,42.690,158.310
C04875=1043.224,368.687,-125.145,173.208,42.695,158.312
C04876=1043.233,368.933,-125.184,173.215,42.699,158.314
C04877=1043.241,369.180,-125.224,173.221,42.703,158.315
C04878=1043.249,369.427,-125.263,173.227,42.707,158.316
C04879=1043.257,369.673,-125.304,173.234,42.712,158.318
C04880=1043.265,369.920,-125.344,173.239,42.716,158.319
C04881=1043.273,370.167,-125.383,173.246,42.720,158.321
C04882=1043.281,370.414,-125.423,173.252,42.725,158.323
C04883=1043.289,370.660,-125.462,173.258,42.729,158.324
C04884=1043.297,370.907,-125.502,173.265,42.733,158.325
C04885=1043.305,371.153,-125.543,173.271,42.738,158.327
C04886=1043.313,371.400,-125.583,173.278,42.742,158.329
C04887=1043.322,371.646,-125.623,173.284,42.747,158.330
C04888=1043.329,371.893,-125.663,173.291,42.751,158.332
C04889=1043.337,372.140,-125.703,173.297,42.756,158.333
C04890=1043.345,372.386,-125.743,173.302,42.760,158.335
C04891=1043.353,372.633,-125.783,173.309,42.764,158.336
C04892=1043.361,372.879,-125.824,173.316,42.770,158.338
C04893=1043.369,373.126,-125.864,173.323,42.774,158.340
C04894=1043.377,373.372,-125.904,173.328,42.778,158.341
C04895=1043.385,373.619,-125.945,173.335,42.783,158.343
C04896=1043.394,373.866,-125.985,173.341,42.787,158.344
C04897=1043.402,374.113,-126.025,173.348,42.792,158.346
C04898=1043.409,374.359,-126.065,173.354,42.797,158.348
C04899=1043.417,374.606,-126.106,173.361,42.801,158.349
C04900=1043.426,374.852,-126.147,173.367,42.806,158.351
C04901=1043.434,375.098,-126.187,173.374,42.810,158.352
C04902=1043.443,375.346,-126.227,173.380,42.815,158.354
C04903=1043.451,375.592,-126.268,173.387,42.820,158.356
C04904=1043.459,375.838,-126.308,173.394,42.824,158.357
C04905=1043.471,376.198,-126.367,173.403,42.831,158.360
C04906=1043.483,376.558,-126.427,173.413,42.838,158.362
C04907=1043.495,376.918,-126.486,173.423,42.845,158.364
C04908=1043.507,377.278,-126.545,173.432,42.852,158.367
C04909=1043.515,377.524,-126.586,173.439,42.856,158.368
C04910=1043.523,377.771,-126.627,173.447,42.861,158.370
C04911=1043.531,378.017,-126.667,173.453,42.866,158.372
C04912=1043.540,378.264,-126.708,173.460,42.871,158.374
C04913=1043.548,378.510,-126.750,173.467,42.875,158.375
C04914=1043.557,378.757,-126.791,173.473,42.880,158.377
C04915=1043.566,379.003,-126.831,173.480,42.885,158.379
C04916=1043.573,379.250,-126.872,173.487,42.890,158.380
C04917=1043.581,379.496,-126.913,173.493,42.895,158.382
C04918=1043.590,379.742,-126.954,173.500,42.899,158.384
C04919=1043.598,379.989,-126.995,173.508,42.904,158.385
C04920=1043.606,380.235,-127.037,173.514,42.909,158.387
C04921=1043.614,380.481,-127.078,173.521,42.914,158.389
C04922=1043.623,380.728,-127.119,173.528,42.919,158.391
C04923=1043.631,380.974,-127.160,173.535,42.924,158.392
C04924=1043.640,381.221,-127.201,173.541,42.929,158.394
C04925=1043.647,381.467,-127.243,173.549,42.934,158.396
C04926=1043.656,381.714,-127.284,173.556,42.939,158.398
C04927=1043.664,381.959,-127.326,173.563,42.944,158.399
C04928=1043.673,382.206,-127.367,173.569,42.949,158.401
C04929=1043.680,382.452,-127.408,173.577,42.954,158.403
C04930=1043.689,382.699,-127.450,173.584,42.959,158.405
C04931=1043.698,382.945,-127.492,173.591,42.964,158.407
C04932=1043.706,383.191,-127.533,173.598,42.969,158.408
C04933=1043.714,383.438,-127.575,173.605,42.974,158.410
C04934=1043.723,383.684,-127.616,173.612,42.979,158.412
C04935=1043.732,383.930,-127.658,173.619,42.984,158.414
C04936=1043.740,384.177,-127.700,173.626,42.990,158.416
C04937=1043.748,384.423,-127.741,173.634,42.994,158.417
C04938=1043.757,384.669,-127.783,173.641,42.999,158.419
C04939=1043.766,384.916,-127.824,173.648,43.005,158.421
C04940=1043.774,385.162,-127.867,173.655,43.010,158.423
C04941=1043.782,385.408,-127.908,173.662,43.015,158.425
C04942=1043.791,385.654,-127.950,173.669,43.020,158.426
C04943=1043.800,385.901,-127.991,173.677,43.026,158.428
C04944=1043.808,386.148,-128.034,173.684,43.031,158.430
C04945=1043.817,386.393,-128.075,173.691,43.036,158.432
C04946=1043.826,386.639,-128.118,173.699,43.041,158.434
C04947=1043.834,386.886,-128.160,173.706,43.046,158.436
C04948=1043.843,387.132,-128.202,173.713,43.052,158.438
C04949=1043.852,387.378,-128.243,173.721,43.057,158.440
C04950=1043.860,387.625,-128.286,173.728,43.062,158.442
C04951=1043.869,387.871,-128.328,173.735,43.067,158.443
C04952=1043.878,388.117,-128.370,173.743,43.073,158.445
C04953=1043.887,388.363,-128.411,173.750,43.078,158.447
C04954=1043.895,388.609,-128.454,173.758,43.083,158.449
C04955=1043.904,388.855,-128.496,173.765,43.089,158.451
C04956=1043.912,389.102,-128.538,173.773,43.094,158.453
C04957=1043.921,389.348,-128.581,173.780,43.100,158.455
C04958=1043.930,389.594,-128.624,173.788,43.105,158.457
C04959=1043.938,389.840,-128.666,173.795,43.110,158.459
C04960=1043.948,390.086,-128.708,173.803,43.116,158.461
C04961=1043.961,390.480,-128.777,173.815,43.125,158.464
C04962=1043.975,390.873,-128.845,173.828,43.133,158.467
C04963=1043.989,391.266,-128.912,173.840,43.142,158.470
C04964=1044.003,391.661,-128.981,173.852,43.151,158.473
C04965=1044.012,391.907,-129.024,173.859,43.157,158.476
C04966=1044.021,392.152,-129.066,173.867,43.162,158.477
C04967=1044.030,392.399,-129.109,173.875,43.168,158.480
C04968=1044.038,392.645,-129.152,173.883,43.174,158.482
C04969=1044.047,392.890,-129.195,173.891,43.179,158.484
C04970=1044.056,393.136,-129.238,173.898,43.185,158.486
C04971=1044.064,393.382,-129.281,173.906,43.191,158.488
C04972=1044.073,393.629,-129.324,173.914,43.197,158.490
C04973=1044.083,393.875,-129.367,173.922,43.202,158.492
C04974=1044.091,394.120,-129.410,173.930,43.208,158.494
C04975=1044.100,394.366,-129.453,173.937,43.214,158.496
C04976=1044.109,394.613,-129.497,173.945,43.220,158.498
C04977=1044.118,394.859,-129.539,173.954,43.225,158.500
C04978=1044.127,395.104,-129.583,173.961,43.231,158.502
C04979=1044.136,395.350,-129.626,173.969,43.237,158.504
C04980=1044.145,395.597,-129.669,173.978,43.242,158.507
C04981=1044.154,395.842,-129.712,173.986,43.248,158.509
C04982=1044.163,396.088,-129.755,173.993,43.254,158.511
C04983=1044.172,396.334,-129.800,174.002,43.260,158.513
C04984=1044.181,396.580,-129.843,174.010,43.266,158.515
C04985=1044.189,396.826,-129.886,174.018,43.272,158.517
C04986=1044.199,397.073,-129.930,174.026,43.278,158.519
C04987=1044.207,397.318,-129.973,174.034,43.284,158.522
C04988=1044.216,397.565,-130.017,174.042,43.290,158.524
C04989=1044.225,397.810,-130.061,174.051,43.296,158.526
C04990=1044.235,398.056,-130.105,174.059,43.302,158.528
C04991=1044.244,398.302,-130.148,174.067,43.308,158.530
C04992=1044.253,398.549,-130.192,174.075,43.314,158.533
C04993=1044.261,398.794,-130.236,174.083,43.320,158.535
C04994=1044.271,399.040,-130.280,174.092,43.326,158.537
C04995=1044.280,399.286,-130.323,174.100,43.332,158.539
C04996=1044.289,399.532,-130.368,174.109,43.339,158.541
C04997=1044.298,399.778,-130.412,174.116,43.344,158.544
C04998=1044.307,400.023,-130.455,174.125,43.351,158.546
C04999=1044.317,400.269,-130.500,174.133,43.357,158.548
C05000=1044.326,400.516,-130.544,174.142,43.363,158.550
C05001=1044.335,400.761,-130.587,174.150,43.369,158.553
C05002=1044.344,401.007,-130.631,174.159,43.375,158.555
C05003=1044.354,401.253,-130.676,174.168,43.381,158.557
C05004=1044.363,401.499,-130.719,174.176,43.388,158.560
C05005=1044.372,401.744,-130.764,174.185,43.394,158.562
C05006=1044.382,401.990,-130.808,174.193,43.400,158.564
C05007=1044.390,402.237,-130.853,174.202,43.406,158.566
C05008=1044.399,402.482,-130.897,174.211,43.413,158.569
C05009=1044.409,402.728,-130.942,174.219,43.419,158.571
C05010=1044.418,402.974,-130.986,174.228,43.426,158.574
C05011=1044.428,403.219,-131.030,174.236,43.432,158.576
C05012=1044.437,403.466,-131.075,174.245,43.438,158.578
C05013=1044.446,403.711,-131.120,174.254,43.445,158.581
C05014=1044.456,403.958,-131.164,174.262,43.451,158.583
C05015=1044.464,404.203,-131.209,174.271,43.458,158.585
C05016=1044.474,404.448,-131.254,174.280,43.464,158.588
C05017=1044.490,404.861,-131.329,174.295,43.475,158.592
C05018=1044.505,405.274,-131.404,174.310,43.486,158.596
C05019=1044.520,405.686,-131.480,174.325,43.497,158.600
C05020=1044.537,406.099,-131.555,174.340,43.509,158.604
C05021=1044.546,406.345,-131.601,174.349,43.515,158.607
C05022=1044.555,406.590,-131.645,174.358,43.522,158.609
C05023=1044.565,406.836,-131.690,174.367,43.528,158.612
C05024=1044.575,407.082,-131.736,174.377,43.535,158.614
C05025=1044.584,407.328,-131.781,174.386,43.542,158.617
C05026=1044.593,407.574,-131.826,174.395,43.549,158.619
C05027=1044.603,407.818,-131.872,174.403,43.555,158.622
C05028=1044.612,408.064,-131.917,174.413,43.562,158.624
C05029=1044.623,408.311,-131.962,174.422,43.569,158.627
C05030=1044.632,408.556,-132.008,174.431,43.576,158.629
C05031=1044.642,408.801,-132.053,174.441,43.582,158.632
C05032=1044.651,409.047,-132.099,174.450,43.589,158.634
C05033=1044.661,409.293,-132.144,174.459,43.596,158.637
C05034=1044.671,409.538,-132.190,174.469,43.603,158.640
C05035=1044.680,409.784,-132.235,174.478,43.610,158.642
C05036=1044.691,410.030,-132.281,174.487,43.616,158.645
C05037=1044.700,410.275,-132.326,174.497,43.624,158.647
C05038=1044.710,410.521,-132.372,174.506,43.630,158.650
C05039=1044.719,410.767,-132.418,174.516,43.638,158.653
C05040=1044.729,411.012,-132.463,174.526,43.644,158.655
C05041=1044.739,411.258,-132.509,174.535,43.651,158.658
C05042=1044.749,411.504,-132.555,174.545,43.658,158.661
C05043=1044.759,411.749,-132.601,174.554,43.665,158.663
C05044=1044.769,411.995,-132.647,174.564,43.672,158.666
C05045=1044.778,412.240,-132.692,174.573,43.680,158.669
C05046=1044.788,412.486,-132.739,174.583,43.687,158.671
C05047=1044.798,412.731,-132.784,174.594,43.694,158.674
C05048=1044.808,412.977,-132.831,174.603,43.701,158.677
C05049=1044.817,413.222,-132.877,174.613,43.708,158.679
C05050=1044.827,413.468,-132.924,174.622,43.715,158.682
C05051=1044.837,413.714,-132.971,174.632,43.723,158.685
C05052=1044.847,413.958,-133.016,174.642,43.730,158.688
C05053=1044.857,414.204,-133.063,174.652,43.737,158.690
C05054=1044.867,414.450,-133.109,174.662,43.745,158.693
C05055=1044.877,414.695,-133.156,174.672,43.752,158.696
C05056=1044.887,414.941,-133.203,174.682,43.759,158.699
C05057=1044.897,415.187,-133.249,174.692,43.766,158.702
C05058=1044.907,415.432,-133.296,174.703,43.774,158.704
C05059=1044.917,415.678,-133.342,174.712,43.781,158.707
C05060=1044.927,415.922,-133.389,174.722,43.789,158.710
C05061=1044.937,416.168,-133.436,174.733,43.796,158.713
C05062=1044.947,416.413,-133.483,174.742,43.804,158.716
C05063=1044.957,416.659,-133.529,174.753,43.811,158.719
C05064=1044.968,416.904,-133.576,174.763,43.819,158.722
C05065=1044.978,417.149,-133.623,174.774,43.826,158.725
C05066=1044.988,417.395,-133.670,174.784,43.834,158.727
C05067=1044.998,417.641,-133.717,174.795,43.842,158.730
C05068=1045.008,417.886,-133.764,174.805,43.849,158.733
C05069=1045.018,418.131,-133.811,174.815,43.857,158.736
C05070=1045.029,418.377,-133.859,174.826,43.864,158.739
C05071=1045.039,418.622,-133.906,174.836,43.872,158.742
C05072=1045.049,418.867,-133.953,174.847,43.879,158.745
C05073=1045.058,419.078,-133.993,174.855,43.886,158.748
C05074=1045.067,419.288,-134.034,174.865,43.893,158.750
C05075=1045.075,419.498,-134.074,174.874,43.899,158.753
C05076=1045.084,419.708,-134.115,174.883,43.907,158.755
C05077=1045.093,419.918,-134.156,174.892,43.913,158.758
C05078=1045.102,420.129,-134.197,174.902,43.920,158.761
C05079=1045.111,420.338,-134.237,174.911,43.926,158.763
C05080=1045.120,420.548,-134.278,174.920,43.933,158.766
C05081=1045.130,420.794,-134.325,174.931,43.941,158.769
C05082=1045.141,421.039,-134.373,174.942,43.949,158.772
C05083=1045.150,421.285,-134.421,174.953,43.957,158.775
C05084=1045.161,421.529,-134.469,174.964,43.965,158.778
C05085=1045.171,421.775,-134.516,174.974,43.973,158.781
C05086=1045.182,422.020,-134.565,174.985,43.981,158.785
C05087=1045.193,422.265,-134.612,174.997,43.989,158.788
C05088=1045.203,422.510,-134.660,175.008,43.997,158.791
C05089=1045.214,422.755,-134.708,175.019,44.005,158.794
C05090=1045.224,423.000,-134.756,175.030,44.013,158.797
C05091=1045.235,423.246,-134.805,175.041,44.021,158.800
C05092=1045.245,423.491,-134.852,175.053,44.029,158.804
C05093=1045.256,423.736,-134.900,175.064,44.037,158.807
C05094=1045.266,423.981,-134.948,175.075,44.046,158.810
C05095=1045.278,424.226,-134.997,175.086,44.054,158.813
C05096=1045.287,424.471,-135.045,175.098,44.062,158.817
C05097=1045.298,424.717,-135.093,175.109,44.070,158.820
C05098=1045.310,424.962,-135.142,175.120,44.078,158.823
C05099=1045.320,425.206,-135.190,175.132,44.087,158.826
C05100=1045.331,425.452,-135.239,175.143,44.095,158.830
C05101=1045.341,425.696,-135.287,175.155,44.104,158.833
C05102=1045.352,425.941,-135.337,175.166,44.112,158.836
C05103=1045.363,426.187,-135.385,175.179,44.120,158.840
C05104=1045.374,426.431,-135.434,175.190,44.129,158.843
C05105=1045.384,426.677,-135.483,175.202,44.137,158.846
C05106=1045.396,426.921,-135.532,175.213,44.146,158.850
C05107=1045.406,427.167,-135.580,175.226,44.154,158.853
C05108=1045.417,427.411,-135.629,175.237,44.163,158.857
C05109=1045.428,427.656,-135.678,175.249,44.171,158.860
C05110=1045.438,427.901,-135.727,175.261,44.180,158.863
C05111=1045.450,428.146,-135.776,175.273,44.188,158.867
C05112=1045.461,428.391,-135.826,175.285,44.197,158.870
C05113=1045.472,428.636,-135.875,175.298,44.206,158.874
C05114=1045.483,428.881,-135.924,175.309,44.214,158.877
C05115=1045.494,429.126,-135.973,175.321,44.223,158.881
C05116=1045.505,429.371,-136.023,175.334,44.232,158.884
C05117=1045.515,429.616,-136.072,175.345,44.241,158.888
C05118=1045.527,429.861,-136.122,175.358,44.250,158.891
C05119=1045.537,430.106,-136.171,175.370,44.259,158.895
C05120=1045.549,430.350,-136.221,175.383,44.268,158.899
C05121=1045.560,430.595,-136.270,175.395,44.277,158.902
C05122=1045.570,430.840,-136.320,175.407,44.285,158.906
C05123=1045.582,431.084,-136.370,175.420,44.295,158.910
C05124=1045.593,431.329,-136.419,175.432,44.303,158.913
C05125=1045.604,431.573,-136.470,175.445,44.313,158.917
C05126=1045.616,431.819,-136.519,175.458,44.321,158.921
C05127=1045.627,432.063,-136.569,175.470,44.331,158.924
C05128=1045.638,432.308,-136.620,175.483,44.340,158.928
C05129=1045.649,432.552,-136.669,175.496,44.348,158.932
C05130=1045.661,432.798,-136.719,175.509,44.358,158.935
C05131=1045.672,433.042,-136.770,175.521,44.367,158.939
C05132=1045.683,433.286,-136.820,175.534,44.376,158.943
C05133=1045.698,433.610,-136.886,175.552,44.388,158.948
C05134=1045.714,433.933,-136.953,175.569,44.400,158.953
C05135=1045.729,434.255,-137.019,175.587,44.413,158.958
C05136=1045.744,434.578,-137.085,175.604,44.425,158.963
C05137=1045.756,434.822,-137.136,175.617,44.434,158.967
C05138=1045.767,435.067,-137.187,175.630,44.444,158.971
C05139=1045.779,435.312,-137.237,175.643,44.453,158.975
C05140=1045.790,435.555,-137.288,175.657,44.463,158.979
C05141=1045.802,435.801,-137.339,175.670,44.472,158.983
C05142=1045.814,436.046,-137.389,175.684,44.482,158.987
C05143=1045.825,436.290,-137.440,175.698,44.491,158.990
C05144=1045.837,436.534,-137.491,175.711,44.501,158.994
C05145=1045.849,436.779,-137.542,175.724,44.510,158.998
C05146=1045.860,437.023,-137.593,175.738,44.520,159.002
C05147=1045.872,437.267,-137.644,175.751,44.530,159.006
C05148=1045.884,437.512,-137.696,175.766,44.540,159.011
C05149=1045.896,437.756,-137.747,175.779,44.549,159.015
C05150=1045.908,438.001,-137.798,175.793,44.559,159.019
C05151=1045.919,438.246,-137.849,175.808,44.569,159.023
C05152=1045.932,438.490,-137.901,175.821,44.579,159.027
C05153=1045.943,438.734,-137.952,175.836,44.588,159.031
C05154=1045.955,438.978,-138.004,175.849,44.598,159.035
C05155=1045.967,439.223,-138.055,175.863,44.608,159.039
C05156=1045.979,439.467,-138.106,175.878,44.618,159.044
C05157=1045.991,439.711,-138.159,175.892,44.628,159.048
C05158=1046.003,439.955,-138.210,175.906,44.638,159.052
C05159=1046.015,440.199,-138.262,175.921,44.648,159.056
C05160=1046.027,440.445,-138.314,175.935,44.658,159.060
C05161=1046.039,440.688,-138.366,175.950,44.668,159.065
C05162=1046.051,440.933,-138.417,175.965,44.678,159.069
C05163=1046.064,441.177,-138.470,175.978,44.688,159.073
C05164=1046.076,441.422,-138.523,175.993,44.699,159.078
C05165=1046.088,441.666,-138.575,176.009,44.709,159.082
C05166=1046.100,441.910,-138.627,176.023,44.719,159.087
C05167=1046.112,442.153,-138.679,176.037,44.729,159.091
C05168=1046.125,442.398,-138.731,176.052,44.739,159.095
C05169=1046.137,442.642,-138.784,176.068,44.750,159.100
C05170=1046.149,442.886,-138.836,176.083,44.760,159.104
C05171=1046.161,443.131,-138.889,176.098,44.771,159.109
C05172=1046.174,443.375,-138.941,176.113,44.781,159.113
C05173=1046.192,443.738,-139.020,176.135,44.797,159.120
C05174=1046.211,444.101,-139.098,176.158,44.812,159.127
C05175=1046.229,444.464,-139.176,176.181,44.828,159.133
C05176=1046.249,444.827,-139.255,176.204,44.844,159.140
C05177=1046.261,445.071,-139.308,176.220,44.854,159.145
C05178=1046.273,445.314,-139.360,176.235,44.865,159.150
C05179=1046.286,445.557,-139.413,176.251,44.876,159.154
C05180=1046.300,445.801,-139.466,176.267,44.886,159.159
C05181=1046.314,446.043,-139.518,176.282,44.897,159.163
C05182=1046.328,446.287,-139.569,176.298,44.907,159.168
C05183=1046.344,446.532,-139.620,176.315,44.917,159.173
C05184=1046.359,446.775,-139.670,176.331,44.927,159.177
C05185=1046.377,447.019,-139.720,176.347,44.937,159.182
C05186=1046.394,447.263,-139.770,176.363,44.947,159.186
C05187=1046.412,447.507,-139.818,176.379,44.956,159.190
C05188=1046.431,447.752,-139.867,176.395,44.966,159.195
C05189=1046.454,448.052,-139.925,176.415,44.978,159.200
C05190=1046.479,448.352,-139.983,176.436,44.989,159.206
C05191=1046.505,448.654,-140.040,176.456,45.000,159.211
C05192=1046.531,448.955,-140.097,176.477,45.011,159.216
C05193=1046.554,449.200,-140.142,176.494,45.020,159.221
C05194=1046.577,449.445,-140.187,176.511,45.028,159.225
C05195=1046.601,449.690,-140.232,176.527,45.037,159.229
C05196=1046.625,449.935,-140.275,176.545,45.045,159.233
C05197=1046.650,450.181,-140.318,176.562,45.054,159.238
C05198=1046.676,450.426,-140.361,176.579,45.062,159.242
C05199=1046.703,450.672,-140.403,176.596,45.069,159.246
C05200=1046.730,450.916,-140.445,176.613,45.078,159.250
C05201=1046.422,450.951,-140.752,176.615,45.163,159.275
C05202=1046.395,450.706,-140.711,176.598,45.155,159.271
C05203=1046.368,450.461,-140.668,176.580,45.147,159.267
C05204=1046.343,450.215,-140.626,176.563,45.139,159.263
C05205=1046.317,449.971,-140.583,176.546,45.131,159.259
C05206=1046.292,449.725,-140.539,176.528,45.123,159.254
C05207=1046.268,449.480,-140.495,176.512,45.114,159.250
C05208=1046.246,449.235,-140.451,176.495,45.105,159.246
C05209=1046.223,448.990,-140.405,176.478,45.097,159.242
C05210=1046.197,448.706,-140.352,176.458,45.087,159.237
C05211=1046.173,448.421,-140.298,176.438,45.076,159.232
C05212=1046.149,448.138,-140.243,176.420,45.066,159.227
C05213=1046.126,447.854,-140.188,176.401,45.055,159.222
C05214=1046.107,447.609,-140.140,176.383,45.046,159.217
C05215=1046.089,447.366,-140.092,176.368,45.037,159.213
C05216=1046.071,447.121,-140.043,176.351,45.027,159.208
C05217=1046.055,446.878,-139.993,176.335,45.017,159.204
C05218=1046.038,446.634,-139.943,176.319,45.007,159.199
C05219=1046.022,446.390,-139.892,176.303,44.997,159.195
C05220=1046.007,446.146,-139.842,176.287,44.987,159.190
C05221=1045.992,445.903,-139.790,176.270,44.977,159.185
C05222=1045.979,445.658,-139.738,176.255,44.966,159.181
C05223=1045.966,445.415,-139.685,176.240,44.956,159.176
C05224=1045.953,445.173,-139.632,176.223,44.946,159.172
C05225=1045.940,444.930,-139.579,176.208,44.935,159.167
C05226=1045.928,444.686,-139.527,176.192,44.924,159.162
C05227=1045.915,444.442,-139.474,176.177,44.914,159.158
C05228=1045.902,444.198,-139.421,176.162,44.903,159.153
C05229=1045.890,443.954,-139.368,176.145,44.893,159.149
C05230=1045.877,443.710,-139.315,176.130,44.883,159.144
C05231=1045.865,443.466,-139.262,176.115,44.872,159.139
C05232=1045.852,443.221,-139.210,176.100,44.862,159.135
C05233=1045.840,442.977,-139.158,176.085,44.852,159.131
C05234=1045.827,442.733,-139.105,176.070,44.841,159.126
C05235=1045.815,442.489,-139.053,176.054,44.831,159.122
C05236=1045.803,442.245,-139.000,176.039,44.821,159.117
C05237=1045.791,442.001,-138.947,176.025,44.810,159.113
C05238=1045.779,441.757,-138.895,176.010,44.800,159.108
C05239=1045.766,441.513,-138.843,175.995,44.790,159.104
C05240=1045.754,441.269,-138.791,175.980,44.780,159.100
C05241=1045.742,441.024,-138.739,175.965,44.770,159.095
C05242=1045.729,440.780,-138.687,175.951,44.760,159.091
C05243=1045.717,440.536,-138.635,175.936,44.749,159.087
C05244=1045.705,440.291,-138.584,175.922,44.740,159.082
C05245=1045.693,440.047,-138.531,175.908,44.730,159.078
C05246=1045.681,439.803,-138.480,175.893,44.720,159.074
C05247=1045.669,439.558,-138.428,175.878,44.710,159.070
C05248=1045.657,439.314,-138.376,175.865,44.700,159.066
C05249=1045.645,439.069,-138.325,175.850,44.690,159.061
C05250=1045.633,438.825,-138.273,175.836,44.680,159.057
C05251=1045.621,438.582,-138.222,175.822,44.671,159.053
C05252=1045.609,438.337,-138.170,175.808,44.661,159.049
C05253=1045.598,438.093,-138.119,175.794,44.651,159.045
C05254=1045.582,437.778,-138.052,175.776,44.639,159.039
C05255=1045.567,437.463,-137.986,175.758,44.626,159.034
C05256=1045.552,437.148,-137.921,175.740,44.614,159.029
C05257=1045.537,436.833,-137.855,175.723,44.601,159.024
C05258=1045.526,436.589,-137.804,175.708,44.592,159.020
C05259=1045.514,436.344,-137.752,175.695,44.583,159.016
C05260=1045.502,436.099,-137.702,175.681,44.573,159.012
C05261=1045.489,435.855,-137.651,175.668,44.563,159.008
C05262=1045.478,435.611,-137.600,175.655,44.554,159.004
C05263=1045.467,435.366,-137.549,175.641,44.545,159.000
C05264=1045.455,435.121,-137.498,175.628,44.535,158.996
C05265=1045.443,434.877,-137.449,175.614,44.526,158.992
C05266=1045.425,434.504,-137.371,175.594,44.512,158.986
C05267=1045.408,434.130,-137.293,175.574,44.498,158.980
C05268=1045.389,433.756,-137.217,175.554,44.484,158.975
C05269=1045.373,433.383,-137.140,175.534,44.469,158.969
C05270=1045.362,433.138,-137.090,175.521,44.460,158.965
C05271=1045.350,432.893,-137.040,175.508,44.452,158.961
C05272=1045.339,432.648,-136.990,175.495,44.442,158.958
C05273=1045.327,432.403,-136.939,175.482,44.433,158.954
C05274=1045.315,432.159,-136.890,175.470,44.424,158.950
C05275=1045.305,431.914,-136.840,175.457,44.415,158.946
C05276=1045.294,431.670,-136.790,175.444,44.406,158.943
C05277=1045.281,431.425,-136.740,175.431,44.398,158.939
C05278=1045.271,431.180,-136.690,175.419,44.388,158.935
C05279=1045.260,430.935,-136.640,175.406,44.379,158.932
C05280=1045.248,430.691,-136.591,175.393,44.371,158.928
C05281=1045.237,430.446,-136.540,175.381,44.361,158.924
C05282=1045.227,430.201,-136.491,175.368,44.353,158.921
C05283=1045.215,429.956,-136.442,175.356,44.344,158.917
C05284=1045.205,429.711,-136.392,175.344,44.335,158.914
C05285=1045.194,429.467,-136.342,175.332,44.326,158.910
C05286=1045.182,429.222,-136.293,175.319,44.318,158.907
C05287=1045.172,428.977,-136.243,175.307,44.309,158.903
C05288=1045.160,428.732,-136.194,175.295,44.301,158.900
C05289=1045.149,428.487,-136.144,175.283,44.292,158.896
C05290=1045.138,428.243,-136.095,175.270,44.283,158.893
C05291=1045.127,427.998,-136.046,175.259,44.275,158.889
C05292=1045.116,427.752,-135.998,175.246,44.266,158.886
C05293=1045.106,427.507,-135.948,175.234,44.257,158.882
C05294=1045.094,427.262,-135.899,175.223,44.249,158.879
C05295=1045.084,427.018,-135.851,175.210,44.241,158.875
C05296=1045.073,426.773,-135.801,175.199,44.232,158.872
C05297=1045.062,426.528,-135.752,175.187,44.223,158.869
C05298=1045.051,426.283,-135.704,175.175,44.215,158.865
C05299=1045.040,426.038,-135.655,175.163,44.207,158.862
C05300=1045.029,425.793,-135.607,175.151,44.198,158.858
C05301=1045.019,425.547,-135.558,175.140,44.191,158.855
C05302=1045.008,425.303,-135.509,175.129,44.182,158.852
C05303=1044.997,425.058,-135.461,175.117,44.174,158.849
C05304=1044.987,424.812,-135.412,175.106,44.165,158.845
C05305=1044.976,424.567,-135.364,175.095,44.157,158.842
C05306=1044.965,424.322,-135.316,175.082,44.149,158.839
C05307=1044.955,424.077,-135.268,175.071,44.141,158.836
C05308=1044.944,423.832,-135.219,175.059,44.133,158.832
C05309=1044.933,423.586,-135.170,175.048,44.125,158.829
C05310=1044.923,423.342,-135.123,175.037,44.117,158.826
C05311=1044.912,423.096,-135.074,175.025,44.108,158.823
C05312=1044.901,422.852,-135.026,175.014,44.100,158.819
C05313=1044.891,422.607,-134.978,175.003,44.092,158.816
C05314=1044.880,422.361,-134.931,174.992,44.085,158.813
C05315=1044.869,422.116,-134.883,174.982,44.076,158.810
C05316=1044.859,421.871,-134.834,174.970,44.068,158.807
C05317=1044.849,421.625,-134.787,174.959,44.060,158.804
C05318=1044.838,421.381,-134.739,174.948,44.052,158.801
C05319=1044.827,421.135,-134.691,174.937,44.045,158.798
C05320=1044.817,420.890,-134.643,174.926,44.037,158.794
C05321=1044.807,420.645,-134.596,174.916,44.029,158.791
C05322=1044.798,420.434,-134.554,174.906,44.022,158.789
C05323=1044.789,420.223,-134.514,174.897,44.016,158.786
C05324=1044.780,420.011,-134.473,174.887,44.009,158.783
C05325=1044.771,419.800,-134.432,174.878,44.002,158.781
C05326=1044.763,419.589,-134.391,174.869,43.995,158.778
C05327=1044.754,419.378,-134.350,174.860,43.989,158.776
C05328=1044.745,419.166,-134.309,174.851,43.982,158.773
C05329=1044.736,418.955,-134.269,174.841,43.976,158.770
C05330=1044.726,418.710,-134.221,174.831,43.968,158.767
C05331=1044.716,418.465,-134.174,174.820,43.960,158.764
C05332=1044.705,418.219,-134.126,174.809,43.953,158.761
C05333=1044.695,417.974,-134.079,174.799,43.945,158.758
C05334=1044.684,417.728,-134.032,174.788,43.938,158.755
C05335=1044.675,417.482,-133.986,174.778,43.930,158.753
C05336=1044.664,417.237,-133.938,174.768,43.923,158.750
C05337=1044.654,416.992,-133.891,174.758,43.915,158.747
C05338=1044.643,416.747,-133.845,174.747,43.908,158.744
C05339=1044.633,416.501,-133.798,174.737,43.900,158.741
C05340=1044.624,416.256,-133.751,174.727,43.893,158.738
C05341=1044.614,416.010,-133.705,174.717,43.885,158.735
C05342=1044.604,415.765,-133.657,174.706,43.878,158.733
C05343=1044.593,415.520,-133.611,174.696,43.871,158.730
C05344=1044.583,415.274,-133.564,174.686,43.864,158.727
C05345=1044.573,415.028,-133.518,174.676,43.856,158.724
C05346=1044.563,414.784,-133.471,174.666,43.849,158.721
C05347=1044.554,414.538,-133.424,174.655,43.841,158.718
C05348=1044.544,414.292,-133.378,174.646,43.834,158.716
C05349=1044.533,414.047,-133.331,174.636,43.827,158.713
C05350=1044.523,413.802,-133.285,174.625,43.820,158.710
C05351=1044.514,413.556,-133.239,174.616,43.813,158.707
C05352=1044.504,413.311,-133.193,174.606,43.806,158.705
C05353=1044.494,413.065,-133.146,174.596,43.799,158.702
C05354=1044.484,412.819,-133.100,174.586,43.791,158.699
C05355=1044.474,412.574,-133.054,174.576,43.784,158.696
C05356=1044.465,412.328,-133.008,174.567,43.777,158.694
C05357=1044.455,412.083,-132.961,174.557,43.770,158.691
C05358=1044.445,411.837,-132.915,174.547,43.763,158.688
C05359=1044.435,411.591,-132.869,174.537,43.756,158.686
C05360=1044.425,411.346,-132.823,174.528,43.749,158.683
C05361=1044.414,411.100,-132.778,174.518,43.742,158.680
C05362=1044.405,410.855,-132.732,174.509,43.735,158.678
C05363=1044.395,410.609,-132.686,174.499,43.728,158.675
C05364=1044.386,410.364,-132.641,174.490,43.721,158.672
C05365=1044.376,410.119,-132.595,174.480,43.715,158.670
C05366=1044.366,409.872,-132.549,174.470,43.707,158.667
C05367=1044.356,409.627,-132.504,174.461,43.701,158.664
C05368=1044.346,409.381,-132.458,174.451,43.694,158.662
C05369=1044.336,409.136,-132.413,174.442,43.687,158.659
C05370=1044.327,408.890,-132.367,174.433,43.681,158.657
C05371=1044.317,408.644,-132.322,174.423,43.673,158.654
C05372=1044.308,408.399,-132.276,174.414,43.667,158.652
C05373=1044.298,408.153,-132.231,174.404,43.660,158.649
C05374=1044.289,407.907,-132.186,174.395,43.653,158.647
C05375=1044.279,407.661,-132.140,174.386,43.647,158.644
C05376=1044.269,407.416,-132.096,174.378,43.640,158.641
C05377=1044.260,407.170,-132.050,174.368,43.633,158.639
C05378=1044.250,406.925,-132.005,174.359,43.627,158.637
C05379=1044.241,406.679,-131.959,174.350,43.620,158.634
C05380=1044.231,406.434,-131.914,174.341,43.613,158.632
C05381=1044.222,406.188,-131.869,174.332,43.607,158.629
C05382=1044.206,405.773,-131.793,174.316,43.596,158.625
C05383=1044.190,405.359,-131.718,174.302,43.585,158.621
C05384=1044.174,404.943,-131.641,174.286,43.574,158.617
C05385=1044.159,404.529,-131.566,174.271,43.563,158.613
C05386=1044.150,404.283,-131.521,174.262,43.557,158.610
C05387=1044.140,404.037,-131.476,174.254,43.550,158.608
C05388=1044.131,403.791,-131.432,174.245,43.543,158.605
C05389=1044.121,403.546,-131.387,174.236,43.537,158.603
C05390=1044.112,403.299,-131.342,174.228,43.531,158.601
C05391=1044.103,403.054,-131.298,174.218,43.525,158.598
C05392=1044.093,402.807,-131.253,174.209,43.518,158.596
C05393=1044.084,402.563,-131.209,174.201,43.512,158.594
C05394=1044.075,402.316,-131.164,174.192,43.506,158.591
C05395=1044.066,402.071,-131.119,174.183,43.500,158.589
C05396=1044.056,401.825,-131.075,174.175,43.493,158.587
C05397=1044.047,401.578,-131.031,174.166,43.487,158.584
